IF bAutoStartPb AND ARbStnBasketAvailibilityRE[8].Q 	THEN ARbStnBasketInActivate[8] 	:= TRUE; ARsStnBasketInTime[8] := DSLocalSystemTimeML.sCurrentDateTime;
ARiStnBasketProductRecipeBuffer[8] 	:= DSStnBasketInfo[8].iProductRecipeNo; ARsStnBasketNoBuffer[8] 	:= DSStnBasketInfo[8].sReservedInt; 	END_IF

IF bAutoStartPb AND ARbStnBasketAvailibilityFE[8].Q 	THEN ARbStnBasketOutActivate[8] 	:= TRUE; ARsStnBasketOutTime[8] := DSLocalSystemTimeML.sCurrentDateTime; 	END_IF

IF bAutoStartPb AND ARbStnBasketAvailibilityRE[9].Q 	THEN ARbStnBasketInActivate[9] 	:= TRUE; ARsStnBasketInTime[9] := DSLocalSystemTimeML.sCurrentDateTime;
ARiStnBasketProductRecipeBuffer[9] 	:= DSStnBasketInfo[9].iProductRecipeNo; ARsStnBasketNoBuffer[9] 	:= DSStnBasketInfo[9].sReservedInt; 	END_IF

IF bAutoStartPb AND ARbStnBasketAvailibilityFE[9].Q 	THEN ARbStnBasketOutActivate[9] 	:= TRUE; ARsStnBasketOutTime[9] := DSLocalSystemTimeML.sCurrentDateTime; 	END_IF

IF bAutoStartPb AND ARbStnBasketAvailibilityRE[10].Q 	THEN ARbStnBasketInActivate[10] 	:= TRUE; ARsStnBasketInTime[10] := DSLocalSystemTimeML.sCurrentDateTime;
ARiStnBasketProductRecipeBuffer[10] 	:= DSStnBasketInfo[10].iProductRecipeNo; ARsStnBasketNoBuffer[10] 	:= DSStnBasketInfo[10].sReservedInt; 	END_IF

IF bAutoStartPb AND ARbStnBasketAvailibilityFE[10].Q 	THEN ARbStnBasketOutActivate[10] 	:= TRUE; ARsStnBasketOutTime[10] := DSLocalSystemTimeML.sCurrentDateTime; 	END_IF

//IF bAutoStartPb AND ARbStnBasketAvailibilityRE[11].Q 	THEN ARbStnBasketInActivate[11] 	:= TRUE; ARsStnBasketInTime[11] := DSLocalSystemTimeML.sCurrentDateTime;
//ARiStnBasketProductRecipeBuffer[11] 	:= DSStnBasketInfo[11].iProductRecipeNo; ARsStnBasketNoBuffer[11] 	:= DSStnBasketInfo[11].sReservedInt; 	END_IF

//IF bAutoStartPb AND ARbStnBasketAvailibilityFE[11].Q 	THEN ARbStnBasketOutActivate[11] 	:= TRUE; ARsStnBasketOutTime[11] := DSLocalSystemTimeML.sCurrentDateTime; 	END_IF

//IF bAutoStartPb AND ARbStnBasketAvailibilityRE[12].Q 	THEN ARbStnBasketInActivate[12] 	:= TRUE; ARsStnBasketInTime[12] := DSLocalSystemTimeML.sCurrentDateTime;
//ARiStnBasketProductRecipeBuffer[12] 	:= DSStnBasketInfo[12].iProductRecipeNo; ARsStnBasketNoBuffer[12] 	:= DSStnBasketInfo[12].sReservedInt; 	END_IF

//IF bAutoStartPb AND ARbStnBasketAvailibilityFE[12].Q 	THEN ARbStnBasketOutActivate[12] 	:= TRUE; ARsStnBasketOutTime[12] := DSLocalSystemTimeML.sCurrentDateTime; 	END_IF



IF bAutoStartPb AND ARtLdNotBasketAvailibility[1].Q 	THEN ARbLdBasketInActivate[1] 	:= FALSE;  	END_IF

IF bAutoStartPb AND ARtUldNotBasketAvailibility[1].Q 	THEN ARbUldBasketInActivate[1] 	:= FALSE; 	END_IF
//IF bAutoStartPb AND ARtUldNotBasketAvailibility[2].Q 	THEN ARbUldBasketInActivate[2] 	:= FALSE; 	END_IF

IF bAutoStartPb AND ARtStnNotBasketAvailibility[1].Q 	THEN ARbStnBasketInActivate[1] 	:= FALSE; 	ARbStnBasketOutActivate[1] 	:= FALSE; 	END_IF
IF bAutoStartPb AND ARtStnNotBasketAvailibility[2].Q 	THEN ARbStnBasketInActivate[2] 	:= FALSE; 	ARbStnBasketOutActivate[2] 	:= FALSE; 	END_IF
IF bAutoStartPb AND ARtStnNotBasketAvailibility[3].Q 	THEN ARbStnBasketInActivate[3] 	:= FALSE; 	ARbStnBasketOutActivate[3] 	:= FALSE; 	END_IF
IF bAutoStartPb AND ARtStnNotBasketAvailibility[4].Q 	THEN ARbStnBasketInActivate[4] 	:= FALSE; 	ARbStnBasketOutActivate[4] 	:= FALSE; 	END_IF
IF bAutoStartPb AND ARtStnNotBasketAvailibility[5].Q 	THEN ARbStnBasketInActivate[5] 	:= FALSE; 	ARbStnBasketOutActivate[5] 	:= FALSE; 	END_IF
IF bAutoStartPb AND ARtStnNotBasketAvailibility[6].Q 	THEN ARbStnBasketInActivate[6] 	:= FALSE; 	ARbStnBasketOutActivate[6] 	:= FALSE; 	END_IF
IF bAutoStartPb AND ARtStnNotBasketAvailibility[7].Q 	THEN ARbStnBasketInActivate[7] 	:= FALSE; 	ARbStnBasketOutActivate[7] 	:= FALSE; 	END_IF
IF bAutoStartPb AND ARtStnNotBasketAvailibility[8].Q 	THEN ARbStnBasketInActivate[8] 	:= FALSE; 	ARbStnBasketOutActivate[8] 	:= FALSE; 	END_IF
IF bAutoStartPb AND ARtStnNotBasketAvailibility[9].Q 	THEN ARbStnBasketInActivate[9] 	:= FALSE; 	ARbStnBasketOutActivate[9] 	:= FALSE; 	END_IF
IF bAutoStartPb AND ARtStnNotBasketAvailibility[10].Q 	THEN ARbStnBasketInActivate[10] 	:= FALSE; 	ARbStnBasketOutActivate[10] 	:= FALSE; 	END_IF
//IF bAutoStartPb AND ARtStnNotBasketAvailibility[11].Q 	THEN ARbStnBasketInActivate[11] 	:= FALSE; 	ARbStnBasketOutActivate[11] 	:= FALSE; 	END_IF
//IF bAutoStartPb AND ARtStnNotBasketAvailibility[12].Q 	THEN ARbStnBasketInActivate[12] 	:= FALSE; 	ARbStnBasketOutActivate[12] 	:= FALSE; 	END_IF

END_PROGRAM

// ---- POUs/MainProgram/DataManagement_Barcode/Log_Configuration.TcPOU
PROGRAM Log_Configuration
VAR
	fb1_dataLog: FB_jx_DataLog;
	fb2_dataLog: FB_jx_DataLog;
	fb3_dataLog: FB_jx_DataLog;
	fb4_dataLog: FB_jx_DataLog;
	fb5_dataLog: FB_jx_DataLog;
	fb6_dataLog: FB_jx_DataLog;
	fb7_dataLog: FB_jx_DataLog;
	fb8_dataLog: FB_jx_DataLog;
	fb9_dataLog: FB_jx_DataLog;
	fb10_dataLog: FB_jx_DataLog;
	(*fb11_dataLog: FB_jx_DataLog;
	fb12_dataLog: FB_jx_DataLog;*)
	fb13_dataLog: FB_jx_DataLog;

	tStn1		: TON;
	tStn2		: TON;
	tStn3		: TON;
	tStn4		: TON;
	tStn5		: TON;
	tStn6		: TON;
	tStn7		: TON;
	tStn8		: TON;
	tStn9		: TON;
	tStn10		: TON;
	tStn11		: TON;
	tStn12		: TON;
	tStn13		: TON;
	uldONtrig	:TON;

	test1		:BOOL;
	test2		:BOOL;
	test3		:BOOL;
	test4		:BOOL;
	test5		:BOOL;
	test6		:BOOL;
	test7		:BOOL;
	test8		:BOOL;
	test9		:BOOL;
	test10		:BOOL;
	test11		:BOOL;
	test12		:BOOL;
	test13		:BOOL;
	test14		:BOOL;
	R_TRIG1	:R_TRIG;
	R_TRIG2	:R_TRIG;
	R_TRIG3	:R_TRIG;

	reset		: BOOL;
	start			: BOOL;
	busy		: BOOL;
	Done		: BOOL;
	write			:BOOL;
	write_done	:BOOL;
	ErrMsg		: STRING;

	tsTimeNow: TIMESTRUCT;


	fbFileRename    : FB_FileRename;
	sNetId          : T_AmsNetId;
        sOldName                : T_MaxString;
        sNewName                : T_MaxString;
        ePath           : E_OpenPath := PATH_GENERIC;          (* Default: generic file path*)
        bExecute                : BOOL;
        tTimeout                : TIME;

	start1: BOOL;
	sPath: STRING;
	sPath1: STRING;
	sNameFile: STRING(255);
	sNameFile1: STRING(255);
	sNameFile2: STRING(255);
	sNameFile3: STRING(255);
	sNameFile4: STRING(255);
	sNameFile5: STRING(255);	(*  *)
	sNameFile6: STRING(255);	(*  *)
	sNameFile7: STRING(255);	(*  *)
	sNameFile8: STRING(255);	(*  *)
	sNameFile9: STRING(255);	(*  *)
	sNameFile10: STRING(255);	(*  *)
	sNameFile11: STRING(255);	(*  *)

	sTimeNow	:STRING;
	RE_BasketCount :R_TRIG;
	iBasketCount:INT;

	bRename: BOOL;
END_VAR

(*
(*All station, only after Remaining timer less than 10 sec, trigger Write CSV*)

tStn1(IN:=ARDsStnSeqProcessCtrl[1].Out_iTotalProcessTimeEV >0 AND ARDsStnSeqProcessCtrl[1].Out_iTotalProcessTimeEV <10 , PT:=T#1s , Q=> , ET=> );
tStn2(IN:=ARDsStnSeqProcessCtrl[2].Out_iTotalProcessTimeEV >0 AND ARDsStnSeqProcessCtrl[2].Out_iTotalProcessTimeEV <10 , PT:=T#1s , Q=> , ET=> );
tStn3(IN:=ARDsStnSeqProcessCtrl[3].Out_iTotalProcessTimeEV >0 AND ARDsStnSeqProcessCtrl[3].Out_iTotalProcessTimeEV <10 , PT:=T#1s , Q=> , ET=> );
tStn4(IN:=ARDsStnSeqProcessCtrl[4].Out_iTotalProcessTimeEV >0 AND ARDsStnSeqProcessCtrl[4].Out_iTotalProcessTimeEV <10  , PT:=T#1s , Q=> , ET=> );
tStn5(IN:=ARDsStnSeqProcessCtrl[5].Out_iTotalProcessTimeEV >0 AND ARDsStnSeqProcessCtrl[5].Out_iTotalProcessTimeEV <10 , PT:=T#1s , Q=> , ET=> );
tStn6(IN:=ARDsStnSeqProcessCtrl[6].Out_iTotalProcessTimeEV >0 AND ARDsStnSeqProcessCtrl[6].Out_iTotalProcessTimeEV <10 , PT:=T#1s , Q=> , ET=> );
tStn7(IN:=ARDsStnSeqProcessCtrl[7].Out_iTotalProcessTimeEV >0 AND ARDsStnSeqProcessCtrl[7].Out_iTotalProcessTimeEV <10 , PT:=T#1s , Q=> , ET=> );
tStn8(IN:=ARDsStnSeqProcessCtrl[8].Out_iTotalProcessTimeEV >0 AND ARDsStnSeqProcessCtrl[8].Out_iTotalProcessTimeEV <10 , PT:=T#1s , Q=> , ET=> );
tStn9(IN:=ARDsStnSeqProcessCtrl[9].Out_iTotalProcessTimeEV >0 AND ARDsStnSeqProcessCtrl[9].Out_iTotalProcessTimeEV <10 , PT:=T#1s, Q=> , ET=> );
tStn10(IN:=ARDsStnSeqProcessCtrl[10].Out_iTotalProcessTimeEV >0 AND ARDsStnSeqProcessCtrl[10].Out_iTotalProcessTimeEV <10 , PT:=T#1s , Q=> , ET=> );
tStn11(IN:=ARDsStnSeqProcessCtrl[11].Out_iTotalProcessTimeEV >0 AND ARDsStnSeqProcessCtrl[11].Out_iTotalProcessTimeEV <10 , PT:=T#1s , Q=> , ET=> );
tStn12(IN:=ARDsStnSeqProcessCtrl[12].Out_iTotalProcessTimeEV >0 AND ARDsStnSeqProcessCtrl[12].Out_iTotalProcessTimeEV <10 , PT:=T#1s , Q=> , ET=> );



(*Create a counter to give a number basket count at the File Name*)

sStn1tittle := CONCAT('-',DSStnBasketInfo[1].ARsBarcodeData[1]);
sStn1tittle := CONCAT(DSStnBasketInfo[1].ARsBarcodeData[2],sStn1tittle);
sStn1tittle := CONCAT('-',sStn1tittle);
sStn1tittle := CONCAT(DSStnBasketInfo[1].ARsBarcodeData[3],sStn1tittle);
sStn1tittle := CONCAT('-',sStn1tittle);
sStn1tittle := CONCAT(DSStnBasketInfo[1].sReservedInt,sStn1tittle);



fb1_dataLog(
	bActivate:= DSStnBasketInfo[1].bAvailibility AND  (tStn1.Q OR GeneratorComparison.ARUpdate_bIntAddress[1]) ,
	FolderDirectory:= 'C:\JKS\report_csv',
	sFileName:= sStn1tittle,
	Tittle := sStn1tittle,
	nNumberOfData:= 50,		(*Max 1000*)
	a_sDataLog_In:= a1_dataLink,
	TimeInterval:= Interval_5s,
	sCsvSeperator:= ',',
	tsTimeNow:=CurrentTime,
	enFIleType:= TXT, 			(*or	 enFIleType:= TXT, 		two option*)
	sMsg=> );


sStn2tittle := CONCAT('-',DSStnBasketInfo[2].ARsBarcodeData[1]);
sStn2tittle := CONCAT(DSStnBasketInfo[2].ARsBarcodeData[2],sStn2tittle);
sStn2tittle := CONCAT('-',sStn2tittle);
sStn2tittle := CONCAT(DSStnBasketInfo[2].ARsBarcodeData[3],sStn2tittle);
sStn2tittle := CONCAT('-',sStn2tittle);
sStn2tittle := CONCAT(DSStnBasketInfo[2].sReservedInt,sStn2tittle);

fb2_dataLog(
	bActivate:= DSStnBasketInfo[2].bAvailibility AND  (tStn2.Q OR GeneratorComparison.ARUpdate_bIntAddress[2]) ,
	FolderDirectory:= 'C:\JKS\report_csv',
	sFileName:= sStn2tittle,
	Tittle := sStn2tittle,
	nNumberOfData:= 50,		(*Max 1000*)
	a_sDataLog_In:= a2_dataLink,
	TimeInterval:= Interval_5s,
	sCsvSeperator:= ',',
	tsTimeNow:=CurrentTime,
	enFIleType:= TXT, 			(*or	 enFIleType:= TXT, 		two option*)
	sMsg=> );


sStn3tittle := CONCAT('-',DSStnBasketInfo[3].ARsBarcodeData[1]);
sStn3tittle := CONCAT(DSStnBasketInfo[3].ARsBarcodeData[2],sStn3tittle);
sStn3tittle := CONCAT('-',sStn3tittle);
sStn3tittle := CONCAT(DSStnBasketInfo[3].ARsBarcodeData[3],sStn3tittle);
sStn3tittle := CONCAT('-',sStn3tittle);
sStn3tittle := CONCAT(DSStnBasketInfo[3].sReservedInt,sStn3tittle);


fb3_dataLog(
	bActivate:= DSStnBasketInfo[3].bAvailibility AND  (tStn3.Q OR GeneratorComparison.ARUpdate_bIntAddress[3]) ,
	FolderDirectory:= 'C:\JKS\report_csv',
	sFileName:= sStn3tittle,
	Tittle := sStn3tittle,
	nNumberOfData:= 50,		(*Max 1000*)
	a_sDataLog_In:= a3_dataLink,
	TimeInterval:= Interval_5s,
	sCsvSeperator:= ',',
	tsTimeNow:=CurrentTime,
	enFIleType:= TXT, 			(*or	 enFIleType:= TXT, 		two option*)
	sMsg=> );


sStn4tittle := CONCAT('-',DSStnBasketInfo[4].ARsBarcodeData[1]);
sStn4tittle := CONCAT(DSStnBasketInfo[4].ARsBarcodeData[2],sStn4tittle);
sStn4tittle := CONCAT('-',sStn4tittle);
sStn4tittle := CONCAT(DSStnBasketInfo[4].ARsBarcodeData[3],sStn4tittle);
sStn4tittle := CONCAT('-',sStn4tittle);
sStn4tittle := CONCAT(DSStnBasketInfo[4].sReservedInt,sStn4tittle);


fb4_dataLog(
	bActivate:= DSStnBasketInfo[4].bAvailibility AND  tStn4.Q ,
	FolderDirectory:= 'C:\JKS\report_csv',
	sFileName:= sStn4tittle,
	Tittle := sStn4tittle,
	nNumberOfData:= 50,		(*Max 1000*)
	a_sDataLog_In:= a4_dataLink,
	TimeInterval:= Interval_5s,
	sCsvSeperator:= ',',
	tsTimeNow:=CurrentTime,
	enFIleType:= TXT, 			(*or	 enFIleType:= TXT, 		two option*)
	sMsg=> );


sStn5tittle := CONCAT('-',DSStnBasketInfo[5].ARsBarcodeData[1]);
sStn5tittle := CONCAT(DSStnBasketInfo[5].ARsBarcodeData[2],sStn5tittle);
sStn5tittle := CONCAT('-',sStn5tittle);
sStn5tittle := CONCAT(DSStnBasketInfo[5].ARsBarcodeData[3],sStn5tittle);
sStn5tittle := CONCAT('-',sStn5tittle);
sStn5tittle := CONCAT(DSStnBasketInfo[5].sReservedInt,sStn5tittle);


fb5_dataLog(
	bActivate:= DSStnBasketInfo[5].bAvailibility AND  (tStn5.Q OR GeneratorComparison.ARUpdate_bIntAddress[5]) ,
	FolderDirectory:= 'C:\JKS\report_csv',
	sFileName:= sStn5tittle,
	Tittle := sStn5tittle,
	nNumberOfData:= 50,		(*Max 1000*)
	a_sDataLog_In:= a5_dataLink,
	TimeInterval:= Interval_5s,
	sCsvSeperator:= ',',
	tsTimeNow:=CurrentTime,
	enFIleType:= TXT, 			(*or	 enFIleType:= TXT, 		two option*)
	sMsg=> );


sStn6tittle := CONCAT('-',DSStnBasketInfo[6].ARsBarcodeData[1]);
sStn6tittle := CONCAT(DSStnBasketInfo[6].ARsBarcodeData[2],sStn6tittle);
sStn6tittle := CONCAT('-',sStn6tittle);
sStn6tittle := CONCAT(DSStnBasketInfo[6].ARsBarcodeData[3],sStn6tittle);
sStn6tittle := CONCAT('-',sStn6tittle);
sStn6tittle := CONCAT(DSStnBasketInfo[6].sReservedInt,sStn6tittle);


fb6_dataLog(
	bActivate:= DSStnBasketInfo[6].bAvailibility AND  tStn6.Q ,
	FolderDirectory:= 'C:\JKS\report_csv',
	sFileName:= sStn6tittle,
	Tittle := sStn6tittle,
	nNumberOfData:= 50,		(*Max 1000*)
	a_sDataLog_In:= a6_dataLink,
	TimeInterval:= Interval_5s,
	sCsvSeperator:= ',',
	tsTimeNow:=CurrentTime,
	enFIleType:= TXT, 			(*or	 enFIleType:= TXT, 		two option*)
	sMsg=> );


sStn7tittle := CONCAT('-',DSStnBasketInfo[7].ARsBarcodeData[1]);
sStn7tittle := CONCAT(DSStnBasketInfo[7].ARsBarcodeData[2],sStn7tittle);
sStn7tittle := CONCAT('-',sStn7tittle);
sStn7tittle := CONCAT(DSStnBasketInfo[7].ARsBarcodeData[3],sStn7tittle);
sStn7tittle := CONCAT('-',sStn7tittle);
sStn7tittle := CONCAT(DSStnBasketInfo[7].sReservedInt,sStn7tittle);

fb7_dataLog(
	bActivate:= DSStnBasketInfo[7].bAvailibility AND  (tStn7.Q OR GeneratorComparison.ARUpdate_bIntAddress[7]) ,
	FolderDirectory:= 'C:\JKS\report_csv',
	sFileName:= sStn7tittle,
	Tittle := sStn7tittle,
	nNumberOfData:= 50,		(*Max 1000*)
	a_sDataLog_In:= a7_dataLink,
	TimeInterval:= Interval_5s,
	sCsvSeperator:= ',',
	tsTimeNow:=CurrentTime,
	enFIleType:= TXT, 			(*or	 enFIleType:= TXT, 		two option*)
	sMsg=> );


sStn8tittle := CONCAT('-',DSStnBasketInfo[8].ARsBarcodeData[1]);
sStn8tittle := CONCAT(DSStnBasketInfo[8].ARsBarcodeData[2],sStn8tittle);
sStn8tittle := CONCAT('-',sStn8tittle);
sStn8tittle := CONCAT(DSStnBasketInfo[8].ARsBarcodeData[3],sStn8tittle);
sStn8tittle := CONCAT('-',sStn8tittle);
sStn8tittle := CONCAT(DSStnBasketInfo[8].sReservedInt,sStn8tittle);

fb8_dataLog(
	bActivate:= DSStnBasketInfo[8].bAvailibility AND  tStn8.Q,
	FolderDirectory:= 'C:\JKS\report_csv',
	sFileName:= sStn8tittle,
	Tittle := sStn8tittle,
	nNumberOfData:= 50,		(*Max 1000*)
	a_sDataLog_In:= a8_dataLink,
	TimeInterval:= Interval_5s,
	sCsvSeperator:= ',',
	tsTimeNow:=CurrentTime,
	enFIleType:= TXT, 			(*or	 enFIleType:= TXT, 		two option*)
	sMsg=> );


sStn9tittle := CONCAT('-',DSStnBasketInfo[9].ARsBarcodeData[1]);
sStn9tittle := CONCAT(DSStnBasketInfo[9].ARsBarcodeData[2],sStn9tittle);
sStn9tittle := CONCAT('-',sStn9tittle);
sStn9tittle := CONCAT(DSStnBasketInfo[9].ARsBarcodeData[3],sStn9tittle);
sStn9tittle := CONCAT('-',sStn9tittle);
sStn9tittle := CONCAT(DSStnBasketInfo[9].sReservedInt,sStn9tittle);

fb9_dataLog(
	bActivate:= DSStnBasketInfo[9].bAvailibility AND  tStn9.Q ,
	FolderDirectory:= 'C:\JKS\report_csv',
	sFileName:= sStn9tittle,
	Tittle := sStn9tittle,
	nNumberOfData:= 50,		(*Max 1000*)
	a_sDataLog_In:= a9_dataLink,
	TimeInterval:= Interval_5s,
	sCsvSeperator:= ',',
	tsTimeNow:=CurrentTime,
	enFIleType:= TXT, 			(*or	 enFIleType:= TXT, 		two option*)
	sMsg=> );


sStn10tittle := CONCAT('-',DSStnBasketInfo[10].ARsBarcodeData[1]);
sStn10tittle := CONCAT(DSStnBasketInfo[10].ARsBarcodeData[2],sStn10tittle);
sStn10tittle := CONCAT('-',sStn10tittle);
sStn10tittle := CONCAT(DSStnBasketInfo[10].ARsBarcodeData[3],sStn10tittle);
sStn10tittle := CONCAT('-',sStn10tittle);
sStn10tittle := CONCAT(DSStnBasketInfo[10].sReservedInt,sStn10tittle);

fb10_dataLog(
	bActivate:=DSStnBasketInfo[10].bAvailibility AND  tStn10.Q,
	FolderDirectory:= 'C:\JKS\report_csv',
	sFileName:= sStn10tittle,
	Tittle := sStn10tittle,
	nNumberOfData:= 50,		(*Max 1000*)
	a_sDataLog_In:= a10_dataLink,
	TimeInterval:= Interval_5s,
	sCsvSeperator:= ',',
	tsTimeNow:=CurrentTime,
	enFIleType:= TXT, 			(*or	 enFIleType:= TXT, 		two option*)
	sMsg=> );

(*
sStn11tittle := CONCAT('-',DSStnBasketInfo[11].ARsBarcodeData[1]);
sStn11tittle := CONCAT(DSStnBasketInfo[11].ARsBarcodeData[2],sStn11tittle);
sStn11tittle := CONCAT('-',sStn11tittle);
sStn11tittle := CONCAT(DSStnBasketInfo[11].ARsBarcodeData[3],sStn11tittle);
sStn11tittle := CONCAT('-',sStn11tittle);
sStn11tittle := CONCAT(DSStnBasketInfo[11].sReservedInt,sStn11tittle);

fb11_dataLog(
	bActivate:=DSStnBasketInfo[11].bAvailibility AND  tStn11.Q ,
	FolderDirectory:= 'C:\JKS\report_csv',
	sFileName:= sStn11tittle,
	Tittle := sStn11tittle,
	nNumberOfData:= 50,		(*Max 1000*)
	a_sDataLog_In:= a11_dataLink,
	TimeInterval:= Interval_5s,
	sCsvSeperator:= ',',
	tsTimeNow:=CurrentTime,
	enFIleType:= TXT, 			(*or	 enFIleType:= TXT, 		two option*)
	sMsg=> );

sStn12tittle := CONCAT('-',DSStnBasketInfo[12].ARsBarcodeData[1]);
sStn12tittle := CONCAT(DSStnBasketInfo[12].ARsBarcodeData[2],sStn12tittle);
sStn12tittle := CONCAT('-',sStn12tittle);
sStn12tittle := CONCAT(DSStnBasketInfo[12].ARsBarcodeData[3],sStn12tittle);
sStn12tittle := CONCAT('-',sStn12tittle);
sStn12tittle := CONCAT(DSStnBasketInfo[12].sReservedInt,sStn12tittle);

fb12_dataLog(
	bActivate:=DSStnBasketInfo[12].bAvailibility AND  tStn12.Q ,
	FolderDirectory:= 'C:\JKS\report_csv',
	sFileName:= sStn12tittle,
	Tittle := sStn12tittle,
	nNumberOfData:= 50,		(*Max 1000*)
	a_sDataLog_In:= a12_dataLink,
	TimeInterval:= Interval_5s,
	sCsvSeperator:= ',',
	tsTimeNow:=CurrentTime,
	enFIleType:= TXT, 			(*or	 enFIleType:= TXT, 		two option*)
	sMsg=> );
*)

(*
sStn13tittle := CONCAT('-',AR2sDSCv_UldConfirmBasketInfo[1,1].ARsBarcodeData[1]);
sStn13tittle := CONCAT(AR2sDSCv_UldConfirmBasketInfo[1,1].ARsBarcodeData[2],sStn13tittle);
sStn13tittle := CONCAT('-',sStn13tittle);
sStn13tittle := CONCAT(AR2sDSCv_UldConfirmBasketInfo[1,1].ARsBarcodeData[3],sStn13tittle);


fb13_dataLog(
	bActivate:= AR2sDSCv_UldConfirmBasketInfo[1,1].bAvailibility (*AND tStn12.Q*) OR test12 (*Trigger Bit when Arm in Down unhook pos*) ,
	FolderDirectory:= 'C:\JKS\report_csv',
	sFileName:= sStn13tittle,
	Tittle := sStn13tittle,
	nNumberOfData:= 50,		(*Max 1000*)
	a_sDataLog_In:= a12_dataLink,
	TimeInterval:= Interval_5s,
	sCsvSeperator:= ',',
	tsTimeNow:=CurrentTime,
	enFIleType:= TXT, 			(*or	 enFIleType:= TXT, 		two option*)
	sMsg=> );
*)

(*To complete the CSV file write at Unloading area*)
IF ARDSArmCtrl[2].AR3sbPositionCfm[3,1,8] OR test14 THEN

	sStn13tittle := CONCAT('-',DSArmBasketInfo[2].ARsBarcodeData[1]);
	sStn13tittle := CONCAT(DSArmBasketInfo[2].ARsBarcodeData[2],sStn13tittle);
	sStn13tittle := CONCAT('-',sStn13tittle);
	sStn13tittle := CONCAT(DSArmBasketInfo[2].ARsBarcodeData[3],sStn13tittle);
	sStn13tittle := CONCAT('-',sStn13tittle);
	sStn13tittle := CONCAT(DSArmBasketInfo[2].sReservedInt,sStn13tittle);

END_IF



(* Trigger bit when Unloading*)
tStn13(IN:=AR2sDSCv_UldConfirmBasketInfo[1,1].bAvailibility , PT:=T#1s , Q=> , ET=> );
R_TRIG1(CLK:=tStn13.Q  OR test13  , Q=> );

	IF R_TRIG1.Q  THEN
		start:=TRUE;
		ELSE
		start:=FALSE;
	END_IF


CurrentTime:=stGetCurrentTime.SysTime;

(*NOTE:-

1-sPath and sPath MUST SAME NAME, otherwise file will not overwrite*)

sPath:=CONCAT('C:\JKS\report_csv','\');
sPath:=CONCAT(sPath,sStn13tittle);
sPath:=CONCAT(sPath,'_');
sPath:=CONCAT(sPath,F_jx_TS_TO_DATE_STRING_1(CurrentTime, '_'));
sPath:=CONCAT(sPath,'.cs_');


sPath1:=CONCAT('C:\JKS\report_csv','\');
sPath1:=CONCAT(sPath1,sStn13tittle);
sPath1:=CONCAT(sPath1,'_');
sPath1:=CONCAT(sPath1,F_jx_TS_TO_DATE_STRING_1(CurrentTime, '_'));
sPath1:=CONCAT(sPath1,'.csv');

fbFileRename(
	sOldName:=sPath ,
	sNewName:=sPath1 ,
	ePath:= PATH_GENERIC,
	bExecute:=bRename OR start);
*)

END_PROGRAM

// ---- FBs/B_JKS_CustomFB/fbDataLogCtrl/FB_jx_DataLog.TcPOU
FUNCTION_BLOCK FB_jx_DataLog
VAR_INPUT
	bActivate:BOOL;		(*Activate data logging*)
	FolderDirectory: T_MaxString;		(*Folder to save log file*)
	Tittle	: T_MaxString;
	sFileName: STRING:='DataLog';
	nNumberOfData:INT:=100;		(*number of data going to log*)
	a_sDataLog_In: ARRAY [1..100] OF ST_DataLog;		(*Log Data name and Value, in string form*)
	TimeInterval: En_TimeInterval:=Interval_1min;		(*Time interval for data logging *)
	sCsvSeperator:STRING:=',';		(*Seperator for Csv file*)
	tsTimeNow: TIMESTRUCT;		(*Time now*)
	enFIleType: En_LogFileType:=CSV;		(*2 Option: CSV ,  TXT*)
	bDirectWrite			: BOOL;
END_VAR
VAR_OUTPUT
	sMsg:STRING;
END_VAR
VAR
	nWriteLogState: INT;
	bTrigWri: BOOL;
	R_TRIG_Wri: R_TRIG;
	a_sDataLog: ARRAY [1..100] OF ST_DataLog;		(*Log Data name and Value, in string form*)
	tsTimeMoment: TIMESTRUCT;
	fbTimeTriggering: FB_TimeTriggering;
	fbWriteLog:FB_WriteLog;
END_VAR

(*
Create by: Jun Xian
Date: 28 May 2014
Modify: 21 Sep 2015

Purpose: 
1. Log data Into Csv file


Feature:
1. Selectable csv seperator.
2. Everyday using a new log file.
3. Selectable data log time interval.
4. Currently number of data support up to 1000 data. 
5. Log File can select save as .CSV or .TXT.

Limitation:
1. If data name > 50, maybe will cause some word missing.
*)
(*
IF bActivate  THEN
fbTimeTriggering(en_interval:= TimeInterval, tsTimeNow:= tsTimeNow, bTrigWriLog=> );
*)
IF bActivate  THEN
bTrigWri := TRUE;
ELSE
bTrigWri := FALSE;
END_IF

R_TRIG_Wri(CLK:= bTrigWri , Q=> );
IF R_TRIG_Wri.Q THEN		(*record the value at that moment*)
a_sDataLog:=a_sDataLog_In;
tsTimeMoment:=tsTimeNow;
END_IF

fbWriteLog(
	sFolderDirectory:= FolderDirectory,
	sTittle := Tittle,
	aDataLog:= a_sDataLog,
	sSeperator:= sCsvSeperator,
	tsTimeMoment:= tsTimeMoment,
	tsTimeNow:= tsTimeNow,
	bStartWri:= R_TRIG_Wri.Q,
	nNumOfData:= nNumberOfData,
	enFileType:= enFIleType,
	sFileName:= sFileName,
	sErrMsg=> sMsg);

END_FUNCTION_BLOCK

// ---- FBs/B_JKS_CustomFB/fbDataLogCtrl/FB_TimeTriggering.TcPOU
FUNCTION_BLOCK FB_TimeTriggering
VAR_INPUT
	en_interval: En_TimeInterval;
	tsTimeNow: TIMESTRUCT;
END_VAR
VAR_OUTPUT
	bTrigWriLog: BOOL;
END_VAR
VAR
	bTest: BOOL;
	wSecPrev: WORD;
END_VAR

IF tsTimeNow.wYear <> 1970 AND tsTimeNow.wYear <> 0 THEN

CASE en_interval OF

Interval_1s:
	IF (tsTimeNow.wSecond <> wSecPrev) THEN
		wSecPrev:=tsTimeNow.wSecond;
		bTrigWriLog:=TRUE;
	ELSE
		bTrigWriLog:=FALSE;
	END_IF

Interval_5s:
	IF (tsTimeNow.wSecond MOD 5 = 0) THEN
		bTrigWriLog:=TRUE;
	ELSE
		bTrigWriLog:=FALSE;
	END_IF

Interval_10s:
	IF (tsTimeNow.wSecond MOD 10 = 0) THEN
		bTrigWriLog:=TRUE;
	ELSE
		bTrigWriLog:=FALSE;
	END_IF

Interval_20s:
	IF (tsTimeNow.wSecond MOD 20 = 0) THEN
	bTrigWriLog:=TRUE;
	ELSE
		bTrigWriLog:=FALSE;
	END_IF

Interval_30s:
	IF (tsTimeNow.wSecond MOD 30 = 0) THEN
	bTrigWriLog:=TRUE;
	ELSE
		bTrigWriLog:=FALSE;
	END_IF

Interval_1min:
	IF (tsTimeNow.wSecond = 0) THEN
	bTrigWriLog:=TRUE;
	ELSE
		bTrigWriLog:=FALSE;
	END_IF

Interval_2min:
	IF (tsTimeNow.wSecond = 0) AND (tsTimeNow.wMinute MOD 2 = 0)THEN
	bTrigWriLog:=TRUE;
	ELSE
		bTrigWriLog:=FALSE;
	END_IF

Interval_5min:
	IF (tsTimeNow.wSecond = 0) AND (tsTimeNow.wMinute MOD 5 = 0)THEN
	bTrigWriLog:=TRUE;
	ELSE
		bTrigWriLog:=FALSE;
	END_IF

Interval_10min:
	IF (tsTimeNow.wSecond = 0) AND (tsTimeNow.wMinute MOD 10 = 0)THEN
	bTrigWriLog:=TRUE;
	ELSE
		bTrigWriLog:=FALSE;
	END_IF

Interval_15min:
	IF (tsTimeNow.wSecond = 0) AND (tsTimeNow.wMinute MOD 15 = 0)THEN
	bTrigWriLog:=TRUE;
	ELSE
		bTrigWriLog:=FALSE;
	END_IF

Interval_20min:
	IF (tsTimeNow.wSecond = 0) AND (tsTimeNow.wMinute MOD 20 = 0)THEN
	bTrigWriLog:=TRUE;
	ELSE
		bTrigWriLog:=FALSE;
	END_IF

Interval_30min:
	IF (tsTimeNow.wSecond = 0) AND (tsTimeNow.wMinute MOD 30 = 0)THEN
	bTrigWriLog:=TRUE;
	ELSE
		bTrigWriLog:=FALSE;
	END_IF

Interval_1h:
	IF (tsTimeNow.wSecond = 0) AND (tsTimeNow.wMinute = 0)THEN
	bTrigWriLog:=TRUE;
	ELSE
		bTrigWriLog:=FALSE;
	END_IF

Interval_2h:
	IF (tsTimeNow.wSecond = 0) AND (tsTimeNow.wMinute = 0) AND (tsTimeNow.wHour MOD 2 = 0)THEN
	bTrigWriLog:=TRUE;
	ELSE
		bTrigWriLog:=FALSE;
	END_IF


END_CASE

END_IF

END_FUNCTION_BLOCK

// ---- FBs/B_JKS_CustomFB/fbDataLogCtrl/FB_WriteLog.TcPOU
FUNCTION_BLOCK FB_WriteLog
VAR_INPUT
	sFolderDirectory: T_MaxString;
	sTittle : T_MaxString;
	aDataLog: ARRAY [1..100] OF ST_DataLog;
	sSeperator: STRING;
	tsTimeMoment: TIMESTRUCT;
	tsTimeNow: TIMESTRUCT;
	bStartWri: BOOL;		(*Been triggered when want start to write log*)
	nNumOfData: INT;
	enFileType: En_LogFileType;
	sFileName: STRING;
	nCurrWrite3: INT;
END_VAR
VAR_OUTPUT
	sErrMsg: STRING;
END_VAR
VAR
	sPath: T_MaxString;
	FB_FileOpen_Log: FB_FileOpen;
	nWriState: INT;
	sHeadline: T_MaxString;
	sHeadline2: T_MaxString;
	i: INT;
	FB_FilePuts_Log: FB_FilePuts;
	sValueLine: T_MaxString;
	FB_FileSeek_Log: FB_FileSeek;
	FB_FileClose_Log: FB_FileClose;
	nCurrWrite: INT := 1;
	bHeadLineDone: BOOL;
	bHeadlineDT: BOOL;
	bHeadlineDT2: BOOL;
	bHeadlineDT3: BOOL;
	bHeadlineDT4: BOOL;
	bDataDT: BOOL;
	bDataDone: BOOL;
	nCurDataWri: INT;
	i_1: INT;
	i_2: INT;
	i_3: INT;
	nCurrWrite2: INT;
	i_4: INT;
	i_5: INT;
	nCurrWrite4: INT;
END_VAR

sPath:=CONCAT(sFolderDirectory,'\');
sPath:=CONCAT(sPath,sFileName);
sPath:=CONCAT(sPath,'_');
sPath:=CONCAT(sPath,F_jx_TS_TO_DATE_STRING_1(tsTimeNow, '_'));
IF enFileType = CSV THEN
	sPath:=CONCAT(sPath,'.csv');
ELSIF enFileType = TXT THEN
	sPath:=CONCAT(sPath,'.cs_');
END_IF

FB_FileOpen_Log(
	sNetId:= ,
	sPathName:= sPath,
	nMode:= ,
	ePath:= PATH_GENERIC,
	bExecute:= ,
	tTimeout:= ,
	bBusy=> ,
	bError=> ,
	nErrId=> ,
	hFile=> );

FB_FilePuts_Log(
	sNetId:= ,
	hFile:= ,
	sLine:= ,
	bExecute:= ,
	tTimeout:= ,
	bBusy=> ,
	bError=> ,
	nErrId=> );

FB_FileSeek_Log(
	sNetId:= ,
	hFile:= ,
	nSeekPos:= ,
	eOrigin:= ,
	bExecute:= ,
	tTimeout:= ,
	bBusy=> ,
	bError=> ,
	nErrId=> );

FB_FileClose_Log(
	sNetId:= ,
	hFile:= ,
	bExecute:= ,
	tTimeout:= ,
	bBusy=> ,
	bError=> ,
	nErrId=> );

Act_WriLogSEQ();

ACTION act_PreapreDataValue:
IF bDataDT THEN
	sValueLine:=F_jx_TS_TO_TIME_STRING(tsTimeMoment);
	sValueLine:=CONCAT(sValueLine,sSeperator);
	(*sValueLine:=CONCAT(sValueLine,F_jx_TS_TO_TIME_STRING(tsTimeMoment));
	sValueLine:=CONCAT(sValueLine,sSeperator);*)
	bDataDT:=FALSE;
	nCurDataWri:=1;

END_IF

FOR i_1:= nCurDataWri TO 1000 DO
	IF i_1 > nNumOfData THEN
		sValueLine:=CONCAT(sValueLine,'$N');
		bDataDone:=TRUE;
EXIT;
	END_IF

	IF ((LEN(sValueLine)+LEN(sSeperator)+LEN(aDataLog[i_1].sValue))<240) THEN		(*T_MaxString is 250, 10 as buffer. the T-MaxString not full yet*)
		sValueLine:=CONCAT(sValueLine,aDataLog[i_1].sValue);
		sValueLine:=CONCAT(sValueLine,sSeperator);
	ELSE		(*T_MaxString is full*)
		bDataDone:=FALSE;
		nCurDataWri:=i_1;
EXIT;	(*T_MaxString is full, write 1st to CSV 1st*)
	END_IF

	IF (i_1 = 1000) THEN	(*Wrtie headline complete*)
		sValueLine:=CONCAT(sValueLine,'$N');
		bDataDone:=TRUE;
EXIT;	(*Write complete*)
	END_IF
END_FOR
END_ACTION

ACTION act_PreparingHeadline:
IF bHeadlineDT THEN		(*new day, need to prepare headline, just come from state 22*)
	(*sHeadline:=sTittle;
	sHeadline:=CONCAT(sHeadline,'$N'); *)


		nCurrWrite4:=1;

		FOR i_5:= nCurrWrite4 TO 7 DO
			IF i_5 > nNumOfData THEN
				sHeadline:=CONCAT(sHeadline,'$N');
				bHeadlineDT:=FALSE;

			EXIT;	(*Write complete*)
			END_IF

			IF ((LEN(sHeadline) + LEN(sSeperator) + LEN(aDataLog[i_5].sName4)) < 240 ) THEN		(*T_MaxString is 250, 10 as buffer. the T-MaxString not full yet*)
				sHeadline:=CONCAT(sHeadline, aDataLog[i_5].sName4);
				sHeadline:=CONCAT(sHeadline,sSeperator);
			ELSE		(*T_MaxString is full*)
				bHeadLineDone:=FALSE;
				nCurrWrite4:=i_5;
			EXIT;	(*T_MaxString is full, write 1st to CSV 1st*)
			END_IF

			IF (i_5 = 7) THEN	(*Wrtie headline complete*)
				sHeadline:=CONCAT(sHeadline,'$N');
				bHeadlineDT:=FALSE;
				bHeadlineDT2:=TRUE;
				nCurrWrite3:=1;
			EXIT;	(*Write complete*)
			END_IF
		END_FOR
END_IF

IF bHeadlineDT2 THEN

		FOR i_4:= nCurrWrite3 TO 7 DO
			IF i_4 > nNumOfData THEN
				sHeadline:=CONCAT(sHeadline,'$N');
				bHeadlineDT2:=FALSE;

			EXIT;	(*Write complete*)
			END_IF

			IF ((LEN(sHeadline) + LEN(sSeperator) + LEN(aDataLog[i_4].sName3)) < 240 ) THEN		(*T_MaxString is 250, 10 as buffer. the T-MaxString not full yet*)
				sHeadline:=CONCAT(sHeadline, aDataLog[i_4].sName3);
				sHeadline:=CONCAT(sHeadline,sSeperator);
			ELSE		(*T_MaxString is full*)
				bHeadLineDone:=FALSE;
				nCurrWrite3:=i_4;
			EXIT;	(*T_MaxString is full, write 1st to CSV 1st*)
			END_IF

			IF (i_4 = 7) THEN	(*Wrtie headline complete*)
				sHeadline:=CONCAT(sHeadline,'$N');
				bHeadlineDT2:=FALSE;
				bHeadlineDT3:=TRUE;
				nCurrWrite2:=1;
			EXIT;	(*Write complete*)
			END_IF
		END_FOR
END_IF

(*sHeadline:=CONCAT(sHeadline,'$N');*)

IF bHeadlineDT3 THEN

		FOR i_3:= nCurrWrite2 TO 50 DO
			IF i_3 > nNumOfData THEN
				sHeadline:=CONCAT(sHeadline,'$N');
				bHeadlineDT3:=FALSE;

			EXIT;	(*Write complete*)
			END_IF

			IF ((LEN(sHeadline) + LEN(sSeperator) + LEN(aDataLog[i_3].sName2)) < 240 ) THEN		(*T_MaxString is 250, 10 as buffer. the T-MaxString not full yet*)
				sHeadline:=CONCAT(sHeadline, aDataLog[i_3].sName2);
				sHeadline:=CONCAT(sHeadline,sSeperator);
			ELSE		(*T_MaxString is full*)
				bHeadLineDone:=FALSE;
				nCurrWrite2:=i_3;
			EXIT;	(*T_MaxString is full, write 1st to CSV 1st*)
			END_IF

			IF (i_3 = 50) THEN	(*Wrtie headline complete*)
				sHeadline:=CONCAT(sHeadline,'$N');
				bHeadlineDT3:=FALSE;
				nCurrWrite:=1;
			EXIT;	(*Write complete*)
			END_IF
		END_FOR

(*sHeadline:=CONCAT(sHeadline,'$N');*)(*comment by syafiq 190418*)

IF NOT (nCurrWrite2=i_3) THEN
	sHeadline:=CONCAT(sHeadline,'Time ');
	sHeadline:=CONCAT(sHeadline,sSeperator);
	bHeadlineDT:=FALSE;
	nCurrWrite:=1;
END_IF

END_IF

FOR i_2:= nCurrWrite TO 1000 DO
	IF i_2 > nNumOfData THEN
		sHeadline:=CONCAT(sHeadline,'$N');
		bHeadLineDone:=TRUE;
EXIT;	(*Write complete*)
	END_IF

	IF ((LEN(sHeadline) + LEN(sSeperator) + LEN(aDataLog[i_2].sName)) < 240 ) THEN		(*T_MaxString is 250, 10 as buffer. the T-MaxString not full yet*)
		sHeadline:=CONCAT(sHeadline, aDataLog[i_2].sName);
		sHeadline:=CONCAT(sHeadline,sSeperator);
	ELSE		(*T_MaxString is full*)
		bHeadLineDone:=FALSE;
		nCurrWrite:=i_2;
EXIT;	(*T_MaxString is full, write 1st to CSV 1st*)
	END_IF

	IF (i_2 = 1000) THEN	(*Wrtie headline complete*)
		sHeadline:=CONCAT(sHeadline,'$N');
		bHeadLineDone:=TRUE;
EXIT;	(*Write complete*)
	END_IF
END_FOR
END_ACTION

ACTION Act_WriLogSEQ:
CASE nWriState OF
0:		(*Iinitial State*)
	FB_FileOpen_Log(bExecute:= FALSE);
	FB_FileSeek_Log(bExecute:= FALSE);
	FB_FilePuts_Log(bExecute:= FALSE);
	FB_FileClose_Log(bExecute:= FALSE);
	
	IF bStartWri THEN
		sErrMsg:='';		(*clear error message*)
(*		bStartWri:=FALSE;*)
		nWriState:=10;
	END_IF

10:		(*Try to write as normal, file already exists*)
	FB_FileOpen_Log(bExecute:= FALSE);
	FB_FileOpen_Log(
		nMode:= FOPEN_MODEREAD OR FOPEN_MODEPLUS OR FOPEN_MODETEXT,
		ePath:= PATH_GENERIC,
		bExecute:= TRUE);

	IF FB_FileOpen_Log.bBusy THEN
		nWriState:=12;
	END_IF

12:		(*Determine whether got error, if error 1804 mean file not exist, need to create a new file*)
	IF NOT FB_FileOpen_Log.bBusy THEN
		IF NOT FB_FileOpen_Log.bError THEN
			nWriState:=14;		(*proceed to write data value*)
		ELSE
			IF (FB_FileOpen_Log.nErrId = 16#70C) THEN		(*no file, need to create a new one*)
			nWriState:=20;
			ELSE
			sErrMsg:='File Open Error [12]';
			nWriState:=0;
			END_IF
		END_IF
	END_IF


14:		(*File Seek, point to the end of file*)
	FB_FileSeek_Log(bExecute:= FALSE);
	FB_FileSeek_Log(
		hFile:= FB_FileOpen_Log.hFile,
		eOrigin:= SEEK_END,
		bExecute:= TRUE);
	
	IF FB_FileSeek_Log.bBusy THEN	(*Seek Fb start to run*)
	nWriState:=16;
	END_IF

16:
	IF NOT FB_FileSeek_Log.bBusy THEN
		IF NOT FB_FileSeek_Log.bError THEN	(*no error*)
bDataDT:=TRUE;
			nWriState:=40;		(*proceed to write *)
		ELSE	(*error*)
			sErrMsg:='File Seek error [16]';
			nWriState:=0;
		END_IF
	END_IF


20:		(*Open a new file, going to write the headline*)
	FB_FileOpen_Log(bExecute:= FALSE);
	FB_FileOpen_Log(
		nMode:= FOPEN_MODEAPPEND OR FOPEN_MODETEXT,
		ePath:= PATH_GENERIC,
		bExecute:= TRUE);
	IF FB_FileOpen_Log.bBusy THEN
		nWriState:=22;
	END_IF

22:		(*check whether got error*)
	IF NOT FB_FileOpen_Log.bBusy  THEN
		IF FB_FileOpen_Log.bError THEN		(*Error*)
			sErrMsg:='File Open error [22]';
			nWriState:=0;
		ELSE		(*no error, go to state 30*)
			nWriState:=30;
bHeadlineDT:=TRUE;
		END_IF

	END_IF


30:		(*Write Headline to Csv	|| Preparing Headline*)
sHeadline:='';
	act_PreparingHeadline();
	FB_FilePuts_Log(bExecute:= FALSE);
	FB_FilePuts_Log(
		hFile:= FB_FileOpen_Log.hFile,
		sLine:= sHeadline,
		bExecute:= TRUE);
	IF FB_FilePuts_Log.bBusy THEN		(*FB start to work*)
		nWriState:=32;
	END_IF

32:
	IF NOT FB_FilePuts_Log.bBusy THEN	(*Fb Done*)
		IF NOT FB_FilePuts_Log.bError THEN	(*no error*)

IF bHeadLineDone THEN	(*Writing headline is complete, can go to write data state*)
nWriState:=40;		(*proceed to write value*)
bDataDT:=TRUE;
ELSE
nWriState:=30;		(*continue to write headline*)
END_IF

		ELSE		(*got error*)
		sErrMsg:='Write Headline Error[32]';
		nWriState:=0;
		END_IF
	END_IF

40:		(*Write data value into csv*)
sValueLine:='';
	act_PreapreDataValue();
	FB_FilePuts_Log(bExecute:= FALSE);
	FB_FilePuts_Log(
		hFile:= FB_FileOpen_Log.hFile,
		sLine:= sValueLine,
		bExecute:= TRUE);
	IF FB_FilePuts_Log.bBusy THEN		(*FB start to work*)
		nWriState:=42;
	END_IF

42:
	IF NOT FB_FilePuts_Log.bBusy THEN
		IF NOT FB_FilePuts_Log.bError THEN	(*no error*)

IF bDataDone THEN		(*write data complete, proceed to close state*)
nWriState:=50;		(*proceed to close file*)
ELSE		(*data not finish write*)
nWriState:=40;		(*continue write data*)
END_IF

		ELSE		(*error*)
			sErrMsg:='Write Value Error[42]';
			nWriState:=0;
		END_IF
	END_IF

50:		(*Close file state*)
	FB_FileClose_Log(bExecute:= FALSE);
	FB_FileClose_Log(
		hFile:= FB_FileOpen_Log.hFile,
		bExecute:= TRUE);
	IF FB_FileClose_Log.bBusy THEN
		nWriState:=52;
	END_IF

52:
	IF NOT FB_FileClose_Log.bBusy THEN
		IF FB_FileClose_Log.bError THEN	(*error*)
		sErrMsg:='File CloseError[52]';
		nWriState:=0;	(*no matter how will goes back to initial state*)
		ELSE	(*no error*)
		nWriState:=0;	(*no matter how will goes back to initial state*)
		END_IF
	END_IF

END_CASE
END_ACTION

END_FUNCTION_BLOCK

// ---- FBs/B_JKS_CustomFB/fbDataLogCtrl/F_jx_TS_TO_DATE_STRING_1.TcPOU
FUNCTION F_jx_TS_TO_DATE_STRING_1 : STRING
VAR_INPUT
	ts_TimeNow: TIMESTRUCT;
	sSeperator: STRING := '/';
END_VAR
VAR
	sDate: STRING;
END_VAR

sDate:='';
sDate:=CONCAT(sDate,WORD_TO_STRING(ts_TimeNow.wYear));
IF ts_TimeNow.wMonth < 10 THEN	(**)
	sDate:=CONCAT(sDate,'0');
	sDate:=CONCAT(sDate,WORD_TO_STRING(ts_TimeNow.wMonth));
ELSE
	sDate:=CONCAT(sDate,WORD_TO_STRING(ts_TimeNow.wMonth));
END_IF

IF ts_TimeNow.wDay < 10 THEN
	sDate:=CONCAT(sDate,'0');
	sDate:=CONCAT(sDate,WORD_TO_STRING(ts_TimeNow.wDay));
ELSE
	sDate:=CONCAT(sDate,WORD_TO_STRING(ts_TimeNow.wDay));
END_IF
F_jx_TS_TO_DATE_STRING_1:=sDate;

END_FUNCTION

// ---- FBs/B_JKS_CustomFB/fbDataLogCtrl/F_jx_TS_TO_TIME_STRING.TcPOU
FUNCTION F_jx_TS_TO_TIME_STRING : STRING
VAR_INPUT
	ts_TimeNow: TIMESTRUCT;
END_VAR
VAR
	sTime:STRING;
	sSeperator: STRING := ':';
END_VAR

sTime:='';
IF ts_TimeNow.wHour < 10 THEN	(*Hour*)
sTime:=CONCAT(sTime,'0');
sTime:=CONCAT(sTime,WORD_TO_STRING(ts_TimeNow.wHour));
ELSE
sTime:=CONCAT(sTime,WORD_TO_STRING(ts_TimeNow.wHour));
END_IF

sTime:=CONCAT(sTime,sSeperator);

IF ts_TimeNow.wMinute < 10 THEN	(*Minute*)
sTime:=CONCAT(sTime,'0');
sTime:=CONCAT(sTime,WORD_TO_STRING(ts_TimeNow.wMinute));
ELSE
sTime:=CONCAT(sTime,WORD_TO_STRING(ts_TimeNow.wMinute));
END_IF

sTime:=CONCAT(sTime,sSeperator);

IF ts_TimeNow.wSecond < 10 THEN	(*Minute*)
sTime:=CONCAT(sTime,'0');
sTime:=CONCAT(sTime,WORD_TO_STRING(ts_TimeNow.wSecond));
ELSE
sTime:=CONCAT(sTime,WORD_TO_STRING(ts_TimeNow.wSecond));
END_IF

F_jx_TS_TO_TIME_STRING:=sTime;

END_FUNCTION

// ---- POUs/MainProgram/DataManagement_Barcode/Log_Management.TcPOU
PROGRAM Log_Management
VAR

END_VAR

;
(*
(*

a2_dataLink[1].sName4:='';
a2_dataLink[2].sName4:='Operator';
a2_dataLink[3].sName4:='Loading ID';
a2_dataLink[4].sName4:='Unloading ID';
a2_dataLink[5].sName4:='Product Recipe Number';
a2_dataLink[6].sName4:='Product Recipe Description';
a2_dataLink[7].sName4:='Load Number';
*)

a1_dataLink[1].sName4:='';
a1_dataLink[2].sName4:='Operator';
a1_dataLink[3].sName4:='LD ID';
a1_dataLink[4].sName4:='ULD ID';
a1_dataLink[5].sName4:='Pro Recipe No';
a1_dataLink[6].sName4:='Pro Recipe Dscrp';
a1_dataLink[7].sName4:='LD No';


a1_dataLink[1].sName3:='';
a1_dataLink[2].sName3:=sUserName;
a1_dataLink[3].sName3:='1';
a1_dataLink[4].sName3:='1';
a1_dataLink[5].sName3:=INT_TO_STRING(DSStnBasketInfo[1].iProductRecipeNo);
a1_dataLink[6].sName3:=DSStnBasketInfo[1].sProgramDescription;
a1_dataLink[7].sName3:=INT_TO_STRING(iProgBatchTotal);


a1_dataLink[1].sName2:='';
a1_dataLink[2].sName2:='N/A';
a1_dataLink[3].sName2:='N/A';
a1_dataLink[4].sName2:='N/A';
a1_dataLink[5].sName2:='N/A';
a1_dataLink[6].sName2:='N/A';
a1_dataLink[7].sName2:='N/A';
a1_dataLink[8].sName2:='Sec';
a1_dataLink[9].sName2:='Sec';
a1_dataLink[10].sName2:='Sec';
a1_dataLink[11].sName2:='Sec';
a1_dataLink[12].sName2:='Sec';
a1_dataLink[13].sName2:='Sec';
a1_dataLink[14].sName2:='DegC';
a1_dataLink[15].sName2:='DegC';
a1_dataLink[16].sName2:='%';
a1_dataLink[17].sName2:='%';
a1_dataLink[18].sName2:='Hz';
a1_dataLink[19].sName2:='Hz';
a1_dataLink[20].sName2:='%';
a1_dataLink[21].sName2:='%';
a1_dataLink[22].sName2:='Hz';
a1_dataLink[23].sName2:='Hz';
a1_dataLink[24].sName2:='%';
a1_dataLink[25].sName2:='%';
a1_dataLink[26].sName2:='Hz';
a1_dataLink[27].sName2:='Hz';
a1_dataLink[28].sName2:='%';
a1_dataLink[29].sName2:='%';
a1_dataLink[30].sName2:='Hz';
a1_dataLink[31].sName2:='Hz';
a1_dataLink[32].sName2:='Kpa';
a1_dataLink[33].sName2:='Kpa';
a1_dataLink[34].sName2:='uS';
a1_dataLink[35].sName2:='uS';
a1_dataLink[36].sName2:='LPM';
a1_dataLink[37].sName2:='LPM';
a1_dataLink[38].sName2:='OHM';
a1_dataLink[39].sName2:='OHM';
a1_dataLink[40].sName2:='PH';
a1_dataLink[41].sName2:='PH';
a1_dataLink[42].sName2:='N/A';
a1_dataLink[43].sName2:='N/A';
a1_dataLink[44].sName2:='Sec';
a1_dataLink[45].sName2:='Sec';


a1_dataLink[1].sName:='Station';
a1_dataLink[2].sName:='Station';
a1_dataLink[3].sName:='Sequences Recipe';
a1_dataLink[4].sName:='Sequences Recipe';
a1_dataLink[5].sName:='Sub Recipe';
a1_dataLink[6].sName:='Sub Recipe';
a1_dataLink[7].sName:='Minimum Time';
a1_dataLink[8].sName:='Minimum Time';
a1_dataLink[9].sName:='Maximum Time';
a1_dataLink[10].sName:='Maximum Time';
a1_dataLink[11].sName:='Effective Time';
a1_dataLink[12].sName:='Effective Time';
a1_dataLink[13].sName:='Temperature';
a1_dataLink[14].sName:='Temperature';
a1_dataLink[15].sName:='U/Sonic Bottom A Power';
a1_dataLink[16].sName:='U/Sonic Bottom A Power';
a1_dataLink[17].sName:='U/Sonic Bottom A Frequency';
a1_dataLink[18].sName:='U/Sonic Bottom A Frequency';
a1_dataLink[19].sName:='U/Sonic Bottom B Power';
a1_dataLink[20].sName:='U/Sonic Bottom B Power';
a1_dataLink[21].sName:='U/Sonic Bottom B Frequency';
a1_dataLink[22].sName:='U/Sonic Bottom B Frequency';
a1_dataLink[23].sName:='U/Sonic Side A Power SV';
a1_dataLink[24].sName:='U/Sonic Side A Power PV';
a1_dataLink[25].sName:='U/Sonic Side A Frequency';
a1_dataLink[26].sName:='U/Sonic Side A Frequency';
a1_dataLink[27].sName:='U/Sonic Side B Power';
a1_dataLink[28].sName:='U/Sonic Side B Power';
a1_dataLink[29].sName:='U/Sonic Side B Frequency';
a1_dataLink[30].sName:='U/Sonic Side B Frequency';
a1_dataLink[31].sName:='Vacuum SV';
a1_dataLink[32].sName:='Vacuum PV';
a1_dataLink[33].sName:='Conductivity';
a1_dataLink[34].sName:='Conductivity';
a1_dataLink[35].sName:='Pump Flow';
a1_dataLink[36].sName:='Pump Flow';
a1_dataLink[37].sName:='Resistivity';
a1_dataLink[38].sName:='Resistivity';
a1_dataLink[39].sName:='PH PV';
a1_dataLink[40].sName:='PH PV';
a1_dataLink[41].sName:='Quality';
a1_dataLink[42].sName:='Quality';
a1_dataLink[43].sName:='Actual Time';
a1_dataLink[44].sName:='Actual Time';


a1_dataLink[1].sValue:='N/A';(*Station*)
a1_dataLink[2].sValue:='1-US Cleaning';(*Station*)
a1_dataLink[3].sValue:='N/A';(*Sequences Recipe*)
a1_dataLink[4].sValue:=DSHmiStationDisplayInfo[1].sStationSequenceRecipeDescription;(*Sequences Recipe*)
a1_dataLink[5].sValue:='N/A';(*Sub Recipe*)
a1_dataLink[6].sValue:=DSHmiStationDisplayInfo[1].sStationSubDescription;(*Sub Recipe*)
a1_dataLink[7].sValue:=INT_TO_STRING(ARDsStnMinMaxEffTimeDisplay[1].iMinTime);(*Minimum Time*)
a1_dataLink[8].sValue:='N/A';(*Minimum Time*)
a1_dataLink[9].sValue:=INT_TO_STRING(ARDsStnMinMaxEffTimeDisplay[1].iMaxTime);(*Maximum Time*)
a1_dataLink[10].sValue:='N/A';(*Maximum Time*)
a1_dataLink[11].sValue:=INT_TO_STRING(ARDsStnMinMaxEffTimeDisplay[1].iEffTime);(*Effective Time*)
a1_dataLink[12].sValue:='N/A';(*Effective Time*)
a1_dataLink[13].sValue:=REAL_TO_STRING(ARrStnTempSV[1]);(*Temperature SV*)
a1_dataLink[14].sValue:=REAL_TO_STRING(ARrStnTempPV[1]);(*Temperature PV*)
a1_dataLink[15].sValue:=INT_TO_STRING(ARiStnManualUSBtmAsv[1]);(*U/Sonic Bottom A Power SV*)
a1_dataLink[16].sValue:=INT_TO_STRING(ARiStnUSBtmAPv[1]);(*U/Sonic Bottom A Power PV*)
a1_dataLink[17].sValue:='N/A';(*U/Sonic Bottom A Frequency SV*)
a1_dataLink[18].sValue:=INT_TO_STRING(DSWeberEnclosure[1].DSWeberGenerator[1].IN_iFreqSetPoint);(*U/Sonic Bottom A Frequency PV*)
a1_dataLink[19].sValue:=INT_TO_STRING(ARiStnManualUSBtmBsv[1]);(*U/Sonic Bottom B Power SV*)
a1_dataLink[20].sValue:=INT_TO_STRING(ARiStnUSBtmBPv[1]);(*U/Sonic Bottom B Power PV*)
a1_dataLink[21].sValue:='N/A';(*U/Sonic Bottom B Frequency SV*)
a1_dataLink[22].sValue:='N/A';(*U/Sonic Bottom B Frequency PV*)
a1_dataLink[23].sValue:='N/A';(*U/Sonic Side A Power SV*)
a1_dataLink[24].sValue:='N/A';(*U/Sonic Side A Power PV*)
a1_dataLink[25].sValue:='N/A';(*U/Sonic Side A Frequency SV*)
a1_dataLink[26].sValue:='N/A';(*U/Sonic Side A Frequency PV*)
a1_dataLink[27].sValue:='N/A';(*U/Sonic Side B Power SV*)
a1_dataLink[28].sValue:='N/A';(*U/Sonic Side B Power PV*)
a1_dataLink[29].sValue:='N/A';(*U/Sonic Side B Frequency SV*)
a1_dataLink[30].sValue:='N/A';(*U/Sonic Side B Frequency PV*)
a1_dataLink[31].sValue:='N/A';(*Vacuum SV*)
a1_dataLink[32].sValue:='N/A';(*Vacuum PV*)
a1_dataLink[33].sValue:='N/A';(*Conductivity SV*)
a1_dataLink[34].sValue:=REAL_TO_STRING(ARrStnConductivityPV[1]);(*Conductivity PV*)
a1_dataLink[35].sValue:='N/A';(*Pump Flow SV*)
a1_dataLink[36].sValue:=REAL_TO_STRING(ARrStnFilterPressurePV[1]);(*Pump Flow PV*)
a1_dataLink[37].sValue:='N/A';(*Resistivity SV*)
a1_dataLink[38].sValue:='N/A';(*Resistivity PV*)
a1_dataLink[39].sValue:='N/A';(*PH SV*)
a1_dataLink[40].sValue:='N/A'; (*PH PV*)
a1_dataLink[41].sValue:='N/A';(*Quality*)
a1_dataLink[42].sValue:=DSStnBasketInfo[1].sProductQuality;(*Quality*)
a1_dataLink[43].sValue:=INT_TO_STRING(ARDsStnSeqProcessCtrl[1].Out_iCurrentProcessTime);(*Actual Time*)
a1_dataLink[44].sValue:='N/A';(*Actual Time*)


(************************************************************************************************************************)

a2_dataLink[1].sName4:='';
a2_dataLink[2].sName4:='Operator';
a2_dataLink[3].sName4:='LD ID';
a2_dataLink[4].sName4:='ULD ID';
a2_dataLink[5].sName4:='Pro Recipe No';
a2_dataLink[6].sName4:='Pro Recipe Dscrp';
a2_dataLink[7].sName4:='LD No';


a2_dataLink[1].sName3:='';
a2_dataLink[2].sName3:=sUserName;
a2_dataLink[3].sName3:='1';
a2_dataLink[4].sName3:='1';
a2_dataLink[5].sName3:=INT_TO_STRING(DSStnBasketInfo[2].iProductRecipeNo);
a2_dataLink[6].sName3:=DSStnBasketInfo[2].sProgramDescription;
a2_dataLink[7].sName3:=INT_TO_STRING(iProgBatchTotal);


a2_dataLink[1].sName2:='';
a2_dataLink[2].sName2:='N/A';
a2_dataLink[3].sName2:='N/A';
a2_dataLink[4].sName2:='N/A';
a2_dataLink[5].sName2:='N/A';
a2_dataLink[6].sName2:='N/A';
a2_dataLink[7].sName2:='N/A';
a2_dataLink[8].sName2:='Sec';
a2_dataLink[9].sName2:='Sec';
a2_dataLink[10].sName2:='Sec';
a2_dataLink[11].sName2:='Sec';
a2_dataLink[12].sName2:='Sec';
a2_dataLink[13].sName2:='Sec';
a2_dataLink[14].sName2:='DegC';
a2_dataLink[15].sName2:='DegC';
a2_dataLink[16].sName2:='%';
a2_dataLink[17].sName2:='%';
a2_dataLink[18].sName2:='Hz';
a2_dataLink[19].sName2:='Hz';
a2_dataLink[20].sName2:='%';
a2_dataLink[21].sName2:='%';
a2_dataLink[22].sName2:='Hz';
a2_dataLink[23].sName2:='Hz';
a2_dataLink[24].sName2:='%';
a2_dataLink[25].sName2:='%';
a2_dataLink[26].sName2:='Hz';
a2_dataLink[27].sName2:='Hz';
a2_dataLink[28].sName2:='%';
a2_dataLink[29].sName2:='%';
a2_dataLink[30].sName2:='Hz';
a2_dataLink[31].sName2:='Hz';
a2_dataLink[32].sName2:='Kpa';
a2_dataLink[33].sName2:='Kpa';
a2_dataLink[34].sName2:='uS';
a2_dataLink[35].sName2:='uS';
a2_dataLink[36].sName2:='LPM';
a2_dataLink[37].sName2:='LPM';
a2_dataLink[38].sName2:='OHM';
a2_dataLink[39].sName2:='OHM';
a2_dataLink[40].sName2:='PH';
a2_dataLink[41].sName2:='PH';
a2_dataLink[42].sName2:='N/A';
a2_dataLink[43].sName2:='N/A';
a2_dataLink[44].sName2:='Sec';
a2_dataLink[45].sName2:='Sec';


a2_dataLink[1].sName:='Station';
a2_dataLink[2].sName:='Station';
a2_dataLink[3].sName:='Sequences Recipe';
a2_dataLink[4].sName:='Sequences Recipe';
a2_dataLink[5].sName:='Sub Recipe';
a2_dataLink[6].sName:='Sub Recipe';
a2_dataLink[7].sName:='Minimum Time';
a2_dataLink[8].sName:='Minimum Time';
a2_dataLink[9].sName:='Maximum Time';
a2_dataLink[10].sName:='Maximum Time';
a2_dataLink[11].sName:='Effective Time';
a2_dataLink[12].sName:='Effective Time';
a2_dataLink[13].sName:='Temperature';
a2_dataLink[14].sName:='Temperature';
a2_dataLink[15].sName:='U/Sonic Bottom A Power';
a2_dataLink[16].sName:='U/Sonic Bottom A Power';
a2_dataLink[17].sName:='U/Sonic Bottom A Frequency';
a2_dataLink[18].sName:='U/Sonic Bottom A Frequency';
a2_dataLink[19].sName:='U/Sonic Bottom B Power';
a2_dataLink[20].sName:='U/Sonic Bottom B Power';
a2_dataLink[21].sName:='U/Sonic Bottom B Frequency';
a2_dataLink[22].sName:='U/Sonic Bottom B Frequency';
a2_dataLink[23].sName:='U/Sonic Side A Power SV';
a2_dataLink[24].sName:='U/Sonic Side A Power PV';
a2_dataLink[25].sName:='U/Sonic Side A Frequency';
a2_dataLink[26].sName:='U/Sonic Side A Frequency';
a2_dataLink[27].sName:='U/Sonic Side B Power';
a2_dataLink[28].sName:='U/Sonic Side B Power';
a2_dataLink[29].sName:='U/Sonic Side B Frequency';
a2_dataLink[30].sName:='U/Sonic Side B Frequency';
a2_dataLink[31].sName:='Vacuum SV';
a2_dataLink[32].sName:='Vacuum PV';
a2_dataLink[33].sName:='Conductivity';
a2_dataLink[34].sName:='Conductivity';
a2_dataLink[35].sName:='Pump Flow';
a2_dataLink[36].sName:='Pump Flow';
a2_dataLink[37].sName:='Resistivity';
a2_dataLink[38].sName:='Resistivity';
a2_dataLink[39].sName:='PH PV';
a2_dataLink[40].sName:='PH PV';
a2_dataLink[41].sName:='Quality';
a2_dataLink[42].sName:='Quality';
a2_dataLink[43].sName:='Actual Time';
a2_dataLink[44].sName:='Actual Time';


a2_dataLink[1].sValue:='N/A';(*Station*)
a2_dataLink[2].sValue:='2-US Cleaning';(*Station*)
a2_dataLink[3].sValue:='N/A';(*Sequences Recipe*)
a2_dataLink[4].sValue:=DSHmiStationDisplayInfo[2].sStationSequenceRecipeDescription;(*Sequences Recipe*)
a2_dataLink[5].sValue:='N/A';(*Sub Recipe*)
a2_dataLink[6].sValue:=DSHmiStationDisplayInfo[2].sStationSubDescription;(*Sub Recipe*)
a2_dataLink[7].sValue:=INT_TO_STRING(ARDsStnMinMaxEffTimeDisplay[2].iMinTime);(*Minimum Time*)
a2_dataLink[8].sValue:='N/A';(*Minimum Time*)
a2_dataLink[9].sValue:=INT_TO_STRING(ARDsStnMinMaxEffTimeDisplay[2].iMaxTime);(*Maximum Time*)
a2_dataLink[10].sValue:='N/A';(*Maximum Time*)
a2_dataLink[11].sValue:=INT_TO_STRING(ARDsStnMinMaxEffTimeDisplay[2].iEffTime);(*Effective Time*)
a2_dataLink[12].sValue:='N/A';(*Effective Time*)
a2_dataLink[13].sValue:=REAL_TO_STRING(ARrStnTempSV[2]);(*Temperature SV*)
a2_dataLink[14].sValue:=REAL_TO_STRING(ARrStnTempPV[2]);(*Temperature PV*)
a2_dataLink[15].sValue:=INT_TO_STRING(ARiStnManualUSBtmAsv[2]);(*U/Sonic Bottom A Power SV*)
a2_dataLink[16].sValue:=INT_TO_STRING(ARiStnUSBtmAPv[2]);(*U/Sonic Bottom A Power PV*)
a2_dataLink[17].sValue:='N/A';(*U/Sonic Bottom A Frequency SV*)
a2_dataLink[18].sValue:=INT_TO_STRING(DSWeberEnclosure[1].DSWeberGenerator[2].IN_iFreqSetPoint);(*U/Sonic Bottom A Frequency PV*)
a2_dataLink[19].sValue:=INT_TO_STRING(ARiStnManualUSBtmBsv[2]);(*U/Sonic Bottom B Power SV*)
a2_dataLink[20].sValue:=INT_TO_STRING(ARiStnUSBtmBPv[2]);(*U/Sonic Bottom B Power PV*)
a2_dataLink[21].sValue:='N/A';(*U/Sonic Bottom B Frequency SV*)
a2_dataLink[22].sValue:='N/A';(*U/Sonic Bottom B Frequency PV*)
a2_dataLink[23].sValue:='N/A';(*U/Sonic Side A Power SV*)
a2_dataLink[24].sValue:='N/A';(*U/Sonic Side A Power PV*)
a2_dataLink[25].sValue:='N/A';(*U/Sonic Side A Frequency SV*)
a2_dataLink[26].sValue:='N/A';(*U/Sonic Side A Frequency PV*)
a2_dataLink[27].sValue:='N/A';(*U/Sonic Side B Power SV*)
a2_dataLink[28].sValue:='N/A';(*U/Sonic Side B Power PV*)
a2_dataLink[29].sValue:='N/A';(*U/Sonic Side B Frequency SV*)
a2_dataLink[30].sValue:='N/A';(*U/Sonic Side B Frequency PV*)
a2_dataLink[31].sValue:='N/A';(*Vacuum SV*)
a2_dataLink[32].sValue:='N/A';(*Vacuum PV*)
a2_dataLink[33].sValue:='N/A';(*Conductivity SV*)
a2_dataLink[34].sValue:=REAL_TO_STRING(ARrStnConductivityPV[2]);(*Conductivity PV*)
a2_dataLink[35].sValue:='N/A';(*Pump Flow SV*)
a2_dataLink[36].sValue:=REAL_TO_STRING(ARrStnFilterPressurePV[2]);(*Pump Flow PV*)
a2_dataLink[37].sValue:='N/A';(*Resistivity SV*)
a2_dataLink[38].sValue:='N/A';(*Resistivity PV*)
a2_dataLink[39].sValue:='N/A';(*PH SV*)
a2_dataLink[40].sValue:='N/A'; (*PH PV*)
a2_dataLink[41].sValue:='N/A';(*Quality*)
a2_dataLink[42].sValue:=DSStnBasketInfo[2].sProductQuality;(*Quality*)
a2_dataLink[43].sValue:=INT_TO_STRING(ARDsStnSeqProcessCtrl[2].Out_iCurrentProcessTime);(*Actual Time*)
a2_dataLink[44].sValue:='N/A';(*Actual Time*)

(************************************************************************************************************************)

a3_dataLink[1].sName4:='';
a3_dataLink[2].sName4:='Operator';
a3_dataLink[3].sName4:='LD ID';
a3_dataLink[4].sName4:='ULD ID';
a3_dataLink[5].sName4:='Pro Recipe No';
a3_dataLink[6].sName4:='Pro Recipe Dscrp';
a3_dataLink[7].sName4:='LD No';


a3_dataLink[1].sName3:='';
a3_dataLink[2].sName3:=sUserName;
a3_dataLink[3].sName3:='1';
a3_dataLink[4].sName3:='1';
a3_dataLink[5].sName3:=INT_TO_STRING(DSStnBasketInfo[3].iProductRecipeNo);
a3_dataLink[6].sName3:=DSStnBasketInfo[3].sProgramDescription;
a3_dataLink[7].sName3:=INT_TO_STRING(iProgBatchTotal);


a3_dataLink[1].sName2:='';
a3_dataLink[2].sName2:='N/A';
a3_dataLink[3].sName2:='N/A';
a3_dataLink[4].sName2:='N/A';
a3_dataLink[5].sName2:='N/A';
a3_dataLink[6].sName2:='N/A';
a3_dataLink[7].sName2:='N/A';
a3_dataLink[8].sName2:='Sec';
a3_dataLink[9].sName2:='Sec';
a3_dataLink[10].sName2:='Sec';
a3_dataLink[11].sName2:='Sec';
a3_dataLink[12].sName2:='Sec';
a3_dataLink[13].sName2:='Sec';
a3_dataLink[14].sName2:='DegC';
a3_dataLink[15].sName2:='DegC';
a3_dataLink[16].sName2:='%';
a3_dataLink[17].sName2:='%';
a3_dataLink[18].sName2:='Hz';
a3_dataLink[19].sName2:='Hz';
a3_dataLink[20].sName2:='%';
a3_dataLink[21].sName2:='%';
a3_dataLink[22].sName2:='Hz';
a3_dataLink[23].sName2:='Hz';
a3_dataLink[24].sName2:='%';
a3_dataLink[25].sName2:='%';
a3_dataLink[26].sName2:='Hz';
a3_dataLink[27].sName2:='Hz';
a3_dataLink[28].sName2:='%';
a3_dataLink[29].sName2:='%';
a3_dataLink[30].sName2:='Hz';
a3_dataLink[31].sName2:='Hz';
a3_dataLink[32].sName2:='Kpa';
a3_dataLink[33].sName2:='Kpa';
a3_dataLink[34].sName2:='uS';
a3_dataLink[35].sName2:='uS';
a3_dataLink[36].sName2:='LPM';
a3_dataLink[37].sName2:='LPM';
a3_dataLink[38].sName2:='OHM';
a3_dataLink[39].sName2:='OHM';
a3_dataLink[40].sName2:='PH';
a3_dataLink[41].sName2:='PH';
a3_dataLink[42].sName2:='N/A';
a3_dataLink[43].sName2:='N/A';
a3_dataLink[44].sName2:='Sec';
a3_dataLink[45].sName2:='Sec';



a3_dataLink[1].sName:='Station';
a3_dataLink[2].sName:='Station';
a3_dataLink[3].sName:='Sequences Recipe';
a3_dataLink[4].sName:='Sequences Recipe';
a3_dataLink[5].sName:='Sub Recipe';
a3_dataLink[6].sName:='Sub Recipe';
a3_dataLink[7].sName:='Minimum Time';
a3_dataLink[8].sName:='Minimum Time';
a3_dataLink[9].sName:='Maximum Time';
a3_dataLink[10].sName:='Maximum Time';
a3_dataLink[11].sName:='Effective Time';
a3_dataLink[12].sName:='Effective Time';
a3_dataLink[13].sName:='Temperature';
a3_dataLink[14].sName:='Temperature';
a3_dataLink[15].sName:='U/Sonic Bottom A Power';
a3_dataLink[16].sName:='U/Sonic Bottom A Power';
a3_dataLink[17].sName:='U/Sonic Bottom A Frequency';
a3_dataLink[18].sName:='U/Sonic Bottom A Frequency';
a3_dataLink[19].sName:='U/Sonic Bottom B Power';
a3_dataLink[20].sName:='U/Sonic Bottom B Power';
a3_dataLink[21].sName:='U/Sonic Bottom B Frequency';
a3_dataLink[22].sName:='U/Sonic Bottom B Frequency';
a3_dataLink[23].sName:='U/Sonic Side A Power SV';
a3_dataLink[24].sName:='U/Sonic Side A Power PV';
a3_dataLink[25].sName:='U/Sonic Side A Frequency';
a3_dataLink[26].sName:='U/Sonic Side A Frequency';
a3_dataLink[27].sName:='U/Sonic Side B Power';
a3_dataLink[28].sName:='U/Sonic Side B Power';
a3_dataLink[29].sName:='U/Sonic Side B Frequency';
a3_dataLink[30].sName:='U/Sonic Side B Frequency';
a3_dataLink[31].sName:='Vacuum SV';
a3_dataLink[32].sName:='Vacuum PV';
a3_dataLink[33].sName:='Conductivity';
a3_dataLink[34].sName:='Conductivity';
a3_dataLink[35].sName:='Pump Flow';
a3_dataLink[36].sName:='Pump Flow';
a3_dataLink[37].sName:='Resistivity';
a3_dataLink[38].sName:='Resistivity';
a3_dataLink[39].sName:='PH PV';
a3_dataLink[40].sName:='PH PV';
a3_dataLink[41].sName:='Quality';
a3_dataLink[42].sName:='Quality';
a3_dataLink[43].sName:='Actual Time';
a3_dataLink[44].sName:='Actual Time';


a3_dataLink[1].sValue:='N/A';(*Station*)
a3_dataLink[2].sValue:='3-US Cleaning';(*Station*)
a3_dataLink[3].sValue:='N/A';(*Sequences Recipe*)
a3_dataLink[4].sValue:=DSHmiStationDisplayInfo[3].sStationSequenceRecipeDescription;(*Sequences Recipe*)
a3_dataLink[5].sValue:='N/A';(*Sub Recipe*)
a3_dataLink[6].sValue:=DSHmiStationDisplayInfo[3].sStationSubDescription;(*Sub Recipe*)
a3_dataLink[7].sValue:=INT_TO_STRING(ARDsStnMinMaxEffTimeDisplay[3].iMinTime);(*Minimum Time*)
a3_dataLink[8].sValue:='N/A';(*Minimum Time*)
a3_dataLink[9].sValue:=INT_TO_STRING(ARDsStnMinMaxEffTimeDisplay[3].iMaxTime);(*Maximum Time*)
a3_dataLink[10].sValue:='N/A';(*Maximum Time*)
a3_dataLink[11].sValue:=INT_TO_STRING(ARDsStnMinMaxEffTimeDisplay[3].iEffTime);(*Effective Time*)
a3_dataLink[12].sValue:='N/A';(*Effective Time*)
a3_dataLink[13].sValue:=REAL_TO_STRING(ARrStnTempSV[3]);(*Temperature SV*)
a3_dataLink[14].sValue:=REAL_TO_STRING(ARrStnTempPV[3]);(*Temperature PV*)
a3_dataLink[15].sValue:=INT_TO_STRING(ARiStnManualUSBtmAsv[3]);(*U/Sonic Bottom A Power SV*)
a3_dataLink[16].sValue:=INT_TO_STRING(ARiStnUSBtmAPv[3]);(*U/Sonic Bottom A Power PV*)
a3_dataLink[17].sValue:='N/A';(*U/Sonic Bottom A Frequency SV*)
a3_dataLink[18].sValue:=INT_TO_STRING(DSWeberEnclosure[1].DSWeberGenerator[3].IN_iFreqSetPoint);(*U/Sonic Bottom A Frequency PV*)
a3_dataLink[19].sValue:=INT_TO_STRING(ARiStnManualUSBtmBsv[3]);(*U/Sonic Bottom B Power SV*)
a3_dataLink[20].sValue:=INT_TO_STRING(ARiStnUSBtmBPv[3]);(*U/Sonic Bottom B Power PV*)
a3_dataLink[21].sValue:='N/A';(*U/Sonic Bottom B Frequency SV*)
a3_dataLink[22].sValue:='N/A';(*U/Sonic Bottom B Frequency PV*)
a3_dataLink[23].sValue:='N/A';(*U/Sonic Side A Power SV*)
a3_dataLink[24].sValue:='N/A';(*U/Sonic Side A Power PV*)
a3_dataLink[25].sValue:='N/A';(*U/Sonic Side A Frequency SV*)
a3_dataLink[26].sValue:='N/A';(*U/Sonic Side A Frequency PV*)
a3_dataLink[27].sValue:='N/A';(*U/Sonic Side B Power SV*)
a3_dataLink[28].sValue:='N/A';(*U/Sonic Side B Power PV*)
a3_dataLink[29].sValue:='N/A';(*U/Sonic Side B Frequency SV*)
a3_dataLink[30].sValue:='N/A';(*U/Sonic Side B Frequency PV*)
a3_dataLink[31].sValue:='N/A';(*Vacuum SV*)
a3_dataLink[32].sValue:='N/A';(*Vacuum PV*)
a3_dataLink[33].sValue:='N/A';(*Conductivity SV*)
a3_dataLink[34].sValue:=REAL_TO_STRING(ARrStnConductivityPV[3]);(*Conductivity PV*)
a3_dataLink[35].sValue:='N/A';(*Pump Flow SV*)
a3_dataLink[36].sValue:=REAL_TO_STRING(ARrStnFilterPressurePV[3]);(*Pump Flow PV*)
a3_dataLink[37].sValue:='N/A';(*Resistivity SV*)
a3_dataLink[38].sValue:='N/A';(*Resistivity PV*)
a3_dataLink[39].sValue:='N/A';(*PH SV*)
a3_dataLink[40].sValue:='N/A'; (*PH PV*)
a3_dataLink[41].sValue:='N/A';(*Quality*)
a3_dataLink[42].sValue:=DSStnBasketInfo[3].sProductQuality;(*Quality*)
a3_dataLink[43].sValue:=INT_TO_STRING(ARDsStnSeqProcessCtrl[3].Out_iCurrentProcessTime);(*Actual Time*)
a3_dataLink[44].sValue:='N/A';(*Actual Time*)

(************************************************************************************************************************)

a4_dataLink[1].sName4:='';
a4_dataLink[2].sName4:='Operator';
a4_dataLink[3].sName4:='LD ID';
a4_dataLink[4].sName4:='ULD ID';
a4_dataLink[5].sName4:='Pro Recipe No';
a4_dataLink[6].sName4:='Pro Recipe Dscrp';
a4_dataLink[7].sName4:='LD No';


a4_dataLink[1].sName3:='';
a4_dataLink[2].sName3:=sUserName;
a4_dataLink[3].sName3:='1';
a4_dataLink[4].sName3:='1';
a4_dataLink[5].sName3:=INT_TO_STRING(DSStnBasketInfo[4].iProductRecipeNo);
a4_dataLink[6].sName3:=DSStnBasketInfo[4].sProgramDescription;
a4_dataLink[7].sName3:=INT_TO_STRING(iProgBatchTotal);


a4_dataLink[1].sName2:='';
a4_dataLink[2].sName2:='N/A';
a4_dataLink[3].sName2:='N/A';
a4_dataLink[4].sName2:='N/A';
a4_dataLink[5].sName2:='N/A';
a4_dataLink[6].sName2:='N/A';
a4_dataLink[7].sName2:='N/A';
a4_dataLink[8].sName2:='Sec';
a4_dataLink[9].sName2:='Sec';
a4_dataLink[10].sName2:='Sec';
a4_dataLink[11].sName2:='Sec';
a4_dataLink[12].sName2:='Sec';
a4_dataLink[13].sName2:='Sec';
a4_dataLink[14].sName2:='DegC';
a4_dataLink[15].sName2:='DegC';
a4_dataLink[16].sName2:='%';
a4_dataLink[17].sName2:='%';
a4_dataLink[18].sName2:='Hz';
a4_dataLink[19].sName2:='Hz';
a4_dataLink[20].sName2:='%';
a4_dataLink[21].sName2:='%';
a4_dataLink[22].sName2:='Hz';
a4_dataLink[23].sName2:='Hz';
a4_dataLink[24].sName2:='%';
a4_dataLink[25].sName2:='%';
a4_dataLink[26].sName2:='Hz';
a4_dataLink[27].sName2:='Hz';
a4_dataLink[28].sName2:='%';
a4_dataLink[29].sName2:='%';
a4_dataLink[30].sName2:='Hz';
a4_dataLink[31].sName2:='Hz';
a4_dataLink[32].sName2:='Kpa';
a4_dataLink[33].sName2:='Kpa';
a4_dataLink[34].sName2:='uS';
a4_dataLink[35].sName2:='uS';
a4_dataLink[36].sName2:='LPM';
a4_dataLink[37].sName2:='LPM';
a4_dataLink[38].sName2:='OHM';
a4_dataLink[39].sName2:='OHM';
a4_dataLink[40].sName2:='PH';
a4_dataLink[41].sName2:='PH';
a4_dataLink[42].sName2:='N/A';
a4_dataLink[43].sName2:='N/A';
a4_dataLink[44].sName2:='Sec';
a4_dataLink[45].sName2:='Sec';


a4_dataLink[1].sName:='Station';
a4_dataLink[2].sName:='Station';
a4_dataLink[3].sName:='Sequences Recipe';
a4_dataLink[4].sName:='Sequences Recipe';
a4_dataLink[5].sName:='Sub Recipe';
a4_dataLink[6].sName:='Sub Recipe';
a4_dataLink[7].sName:='Minimum Time';
a4_dataLink[8].sName:='Minimum Time';
a4_dataLink[9].sName:='Maximum Time';
a4_dataLink[10].sName:='Maximum Time';
a4_dataLink[11].sName:='Effective Time';
a4_dataLink[12].sName:='Effective Time';
a4_dataLink[13].sName:='Temperature';
a4_dataLink[14].sName:='Temperature';
a4_dataLink[15].sName:='U/Sonic Bottom A Power';
a4_dataLink[16].sName:='U/Sonic Bottom A Power';
a4_dataLink[17].sName:='U/Sonic Bottom A Frequency';
a4_dataLink[18].sName:='U/Sonic Bottom A Frequency';
a4_dataLink[19].sName:='U/Sonic Bottom B Power';
a4_dataLink[20].sName:='U/Sonic Bottom B Power';
a4_dataLink[21].sName:='U/Sonic Bottom B Frequency';
a4_dataLink[22].sName:='U/Sonic Bottom B Frequency';
a4_dataLink[23].sName:='U/Sonic Side A Power SV';
a4_dataLink[24].sName:='U/Sonic Side A Power PV';
a4_dataLink[25].sName:='U/Sonic Side A Frequency';
a4_dataLink[26].sName:='U/Sonic Side A Frequency';
a4_dataLink[27].sName:='U/Sonic Side B Power';
a4_dataLink[28].sName:='U/Sonic Side B Power';
a4_dataLink[29].sName:='U/Sonic Side B Frequency';
a4_dataLink[30].sName:='U/Sonic Side B Frequency';
a4_dataLink[31].sName:='Vacuum SV';
a4_dataLink[32].sName:='Vacuum PV';
a4_dataLink[33].sName:='Conductivity';
a4_dataLink[34].sName:='Conductivity';
a4_dataLink[35].sName:='Pump Flow';
a4_dataLink[36].sName:='Pump Flow';
a4_dataLink[37].sName:='Resistivity';
a4_dataLink[38].sName:='Resistivity';
a4_dataLink[39].sName:='PH PV';
a4_dataLink[40].sName:='PH PV';
a4_dataLink[41].sName:='Quality';
a4_dataLink[42].sName:='Quality';
a4_dataLink[43].sName:='Actual Time';
a4_dataLink[44].sName:='Actual Time';


a4_dataLink[1].sValue:='N/A';(*Station*)
a4_dataLink[2].sValue:='4-Rinsing';(*Station*)
a4_dataLink[3].sValue:='N/A';(*Sequences Recipe*)
a4_dataLink[4].sValue:=DSHmiStationDisplayInfo[4].sStationSequenceRecipeDescription;(*Sequences Recipe*)
a4_dataLink[5].sValue:='N/A';(*Sub Recipe*)
a4_dataLink[6].sValue:=DSHmiStationDisplayInfo[4].sStationSubDescription;(*Sub Recipe*)
a4_dataLink[7].sValue:=INT_TO_STRING(ARDsStnMinMaxEffTimeDisplay[4].iMinTime);(*Minimum Time*)
a4_dataLink[8].sValue:='N/A';(*Minimum Time*)
a4_dataLink[9].sValue:=INT_TO_STRING(ARDsStnMinMaxEffTimeDisplay[4].iMaxTime);(*Maximum Time*)
a4_dataLink[10].sValue:='N/A';(*Maximum Time*)
a4_dataLink[11].sValue:=INT_TO_STRING(ARDsStnMinMaxEffTimeDisplay[4].iEffTime);(*Effective Time*)
a4_dataLink[12].sValue:='N/A';(*Effective Time*)
a4_dataLink[13].sValue:=REAL_TO_STRING(ARrStnTempSV[4]);(*Temperature SV*)
a4_dataLink[14].sValue:=REAL_TO_STRING(ARrStnTempPV[4]);(*Temperature PV*)
a4_dataLink[15].sValue:=INT_TO_STRING(ARiStnManualUSBtmAsv[4]);(*U/Sonic Bottom A Power SV*)
a4_dataLink[16].sValue:=INT_TO_STRING(ARiStnUSBtmAPv[4]);(*U/Sonic Bottom A Power PV*)
a4_dataLink[17].sValue:='N/A';(*U/Sonic Bottom A Frequency SV*)
a4_dataLink[18].sValue:='N/A';(*U/Sonic Bottom A Frequency PV*)
a4_dataLink[19].sValue:=INT_TO_STRING(ARiStnManualUSBtmBsv[4]);(*U/Sonic Bottom B Power SV*)
a4_dataLink[20].sValue:=INT_TO_STRING(ARiStnUSBtmBPv[4]);(*U/Sonic Bottom B Power PV*)
a4_dataLink[21].sValue:='N/A';(*U/Sonic Bottom B Frequency SV*)
a4_dataLink[22].sValue:='N/A';(*U/Sonic Bottom B Frequency PV*)
a4_dataLink[23].sValue:='N/A';(*U/Sonic Side A Power SV*)
a4_dataLink[24].sValue:='N/A';(*U/Sonic Side A Power PV*)
a4_dataLink[25].sValue:='N/A';(*U/Sonic Side A Frequency SV*)
a4_dataLink[26].sValue:='N/A';(*U/Sonic Side A Frequency PV*)
a4_dataLink[27].sValue:='N/A';(*U/Sonic Side B Power SV*)
a4_dataLink[28].sValue:='N/A';(*U/Sonic Side B Power PV*)
a4_dataLink[29].sValue:='N/A';(*U/Sonic Side B Frequency SV*)
a4_dataLink[30].sValue:='N/A';(*U/Sonic Side B Frequency PV*)
a4_dataLink[31].sValue:='N/A';(*Vacuum SV*)
a4_dataLink[32].sValue:='N/A';(*Vacuum PV*)
a4_dataLink[33].sValue:='N/A';(*Conductivity SV*)
a4_dataLink[34].sValue:=REAL_TO_STRING(ARrStnConductivityPV[4]);(*Conductivity PV*)
a4_dataLink[35].sValue:='N/A';(*Pump Flow SV*)
a4_dataLink[36].sValue:=REAL_TO_STRING(ARrStnFilterPressurePV[4]);(*Pump Flow PV*)
a4_dataLink[37].sValue:='N/A';(*Resistivity SV*)
a4_dataLink[38].sValue:='N/A';(*Resistivity PV*)
a4_dataLink[39].sValue:='N/A';(*PH SV*)
a4_dataLink[40].sValue:='N/A'; (*PH PV*)
a4_dataLink[41].sValue:='N/A';(*Quality*)
a4_dataLink[42].sValue:=DSStnBasketInfo[4].sProductQuality;(*Quality*)
a4_dataLink[43].sValue:=INT_TO_STRING(ARDsStnSeqProcessCtrl[4].Out_iCurrentProcessTime);(*Actual Time*)
a4_dataLink[44].sValue:='N/A';(*Actual Time*)

(************************************************************************************************************************)
a5_dataLink[1].sName4:='';
a5_dataLink[2].sName4:='Operator';
a5_dataLink[3].sName4:='LD ID';
a5_dataLink[4].sName4:='ULD ID';
a5_dataLink[5].sName4:='Pro Recipe No';
a5_dataLink[6].sName4:='Pro Recipe Dscrp';
a5_dataLink[7].sName4:='LD No';


a5_dataLink[1].sName3:='';
a5_dataLink[2].sName3:=sUserName;
a5_dataLink[3].sName3:='1';
a5_dataLink[4].sName3:='1';
a5_dataLink[5].sName3:=INT_TO_STRING(DSStnBasketInfo[5].iProductRecipeNo);
a5_dataLink[6].sName3:=DSStnBasketInfo[5].sProgramDescription;
a5_dataLink[7].sName3:=INT_TO_STRING(iProgBatchTotal);

a5_dataLink[1].sName2:='';
a5_dataLink[2].sName2:='N/A';
a5_dataLink[3].sName2:='N/A';
a5_dataLink[4].sName2:='N/A';
a5_dataLink[5].sName2:='N/A';
a5_dataLink[6].sName2:='N/A';
a5_dataLink[7].sName2:='N/A';
a5_dataLink[8].sName2:='Sec';
a5_dataLink[9].sName2:='Sec';
a5_dataLink[10].sName2:='Sec';
a5_dataLink[11].sName2:='Sec';
a5_dataLink[12].sName2:='Sec';
a5_dataLink[13].sName2:='Sec';
a5_dataLink[14].sName2:='DegC';
a5_dataLink[15].sName2:='DegC';
a5_dataLink[16].sName2:='%';
a5_dataLink[17].sName2:='%';
a5_dataLink[18].sName2:='Hz';
a5_dataLink[19].sName2:='Hz';
a5_dataLink[20].sName2:='%';
a5_dataLink[21].sName2:='%';
a5_dataLink[22].sName2:='Hz';
a5_dataLink[23].sName2:='Hz';
a5_dataLink[24].sName2:='%';
a5_dataLink[25].sName2:='%';
a5_dataLink[26].sName2:='Hz';
a5_dataLink[27].sName2:='Hz';
a5_dataLink[28].sName2:='%';
a5_dataLink[29].sName2:='%';
a5_dataLink[30].sName2:='Hz';
a5_dataLink[31].sName2:='Hz';
a5_dataLink[32].sName2:='Kpa';
a5_dataLink[33].sName2:='Kpa';
a5_dataLink[34].sName2:='uS';
a5_dataLink[35].sName2:='uS';
a5_dataLink[36].sName2:='LPM';
a5_dataLink[37].sName2:='LPM';
a5_dataLink[38].sName2:='OHM';
a5_dataLink[39].sName2:='OHM';
a5_dataLink[40].sName2:='PH';
a5_dataLink[41].sName2:='PH';
a5_dataLink[42].sName2:='N/A';
a5_dataLink[43].sName2:='N/A';
a5_dataLink[44].sName2:='Sec';
a5_dataLink[45].sName2:='Sec';



a5_dataLink[1].sName:='Station';
a5_dataLink[2].sName:='Station';
a5_dataLink[3].sName:='Sequences Recipe';
a5_dataLink[4].sName:='Sequences Recipe';
a5_dataLink[5].sName:='Sub Recipe';
a5_dataLink[6].sName:='Sub Recipe';
a5_dataLink[7].sName:='Minimum Time';
a5_dataLink[8].sName:='Minimum Time';
a5_dataLink[9].sName:='Maximum Time';
a5_dataLink[10].sName:='Maximum Time';
a5_dataLink[11].sName:='Effective Time';
a5_dataLink[12].sName:='Effective Time';
a5_dataLink[13].sName:='Temperature';
a5_dataLink[14].sName:='Temperature';
a5_dataLink[15].sName:='U/Sonic Bottom A Power';
a5_dataLink[16].sName:='U/Sonic Bottom A Power';
a5_dataLink[17].sName:='U/Sonic Bottom A Frequency';
a5_dataLink[18].sName:='U/Sonic Bottom A Frequency';
a5_dataLink[19].sName:='U/Sonic Bottom B Power';
a5_dataLink[20].sName:='U/Sonic Bottom B Power';
a5_dataLink[21].sName:='U/Sonic Bottom B Frequency';
a5_dataLink[22].sName:='U/Sonic Bottom B Frequency';
a5_dataLink[23].sName:='U/Sonic Side A Power SV';
a5_dataLink[24].sName:='U/Sonic Side A Power PV';
a5_dataLink[25].sName:='U/Sonic Side A Frequency';
a5_dataLink[26].sName:='U/Sonic Side A Frequency';
a5_dataLink[27].sName:='U/Sonic Side B Power';
a5_dataLink[28].sName:='U/Sonic Side B Power';
a5_dataLink[29].sName:='U/Sonic Side B Frequency';
a5_dataLink[30].sName:='U/Sonic Side B Frequency';
a5_dataLink[31].sName:='Vacuum SV';
a5_dataLink[32].sName:='Vacuum PV';
a5_dataLink[33].sName:='Conductivity';
a5_dataLink[34].sName:='Conductivity';
a5_dataLink[35].sName:='Pump Flow';
a5_dataLink[36].sName:='Pump Flow';
a5_dataLink[37].sName:='Resistivity';
a5_dataLink[38].sName:='Resistivity';
a5_dataLink[39].sName:='PH PV';
a5_dataLink[40].sName:='PH PV';
a5_dataLink[41].sName:='Quality';
a5_dataLink[42].sName:='Quality';
a5_dataLink[43].sName:='Actual Time';
a5_dataLink[44].sName:='Actual Time';


a5_dataLink[1].sValue:='N/A';(*Station*)
a5_dataLink[2].sValue:='5-US Cleaning';(*Station*)
a5_dataLink[3].sValue:='N/A';(*Sequences Recipe*)
a5_dataLink[4].sValue:=DSHmiStationDisplayInfo[5].sStationSequenceRecipeDescription;(*Sequences Recipe*)
a5_dataLink[5].sValue:='N/A';(*Sub Recipe*)
a5_dataLink[6].sValue:=DSHmiStationDisplayInfo[5].sStationSubDescription;(*Sub Recipe*)
a5_dataLink[7].sValue:=INT_TO_STRING(ARDsStnMinMaxEffTimeDisplay[5].iMinTime);(*Minimum Time*)
a5_dataLink[8].sValue:='N/A';(*Minimum Time*)
a5_dataLink[9].sValue:=INT_TO_STRING(ARDsStnMinMaxEffTimeDisplay[5].iMaxTime);(*Maximum Time*)
a5_dataLink[10].sValue:='N/A';(*Maximum Time*)
a5_dataLink[11].sValue:=INT_TO_STRING(ARDsStnMinMaxEffTimeDisplay[5].iEffTime);(*Effective Time*)
a5_dataLink[12].sValue:='N/A';(*Effective Time*)
a5_dataLink[13].sValue:=REAL_TO_STRING(ARrStnTempSV[5]);(*Temperature SV*)
a5_dataLink[14].sValue:=REAL_TO_STRING(ARrStnTempPV[5]);(*Temperature PV*)
a5_dataLink[15].sValue:=INT_TO_STRING(ARiStnManualUSBtmAsv[5]);(*U/Sonic Bottom A Power SV*)
a5_dataLink[16].sValue:=INT_TO_STRING(ARiStnUSBtmAPv[5]);(*U/Sonic Bottom A Power PV*)
a5_dataLink[17].sValue:='N/A';(*U/Sonic Bottom A Frequency SV*)
a5_dataLink[18].sValue:=INT_TO_STRING(DSWeberEnclosure[1].DSWeberGenerator[5].IN_iFreqSetPoint);(*U/Sonic Bottom A Frequency PV*)
a5_dataLink[19].sValue:=INT_TO_STRING(ARiStnManualUSBtmBsv[5]);(*U/Sonic Bottom B Power SV*)
a5_dataLink[20].sValue:=INT_TO_STRING(ARiStnUSBtmBPv[5]);(*U/Sonic Bottom B Power PV*)
a5_dataLink[21].sValue:='N/A';(*U/Sonic Bottom B Frequency SV*)
a5_dataLink[22].sValue:='N/A';(*U/Sonic Bottom B Frequency PV*)
a5_dataLink[23].sValue:='N/A';(*U/Sonic Side A Power SV*)
a5_dataLink[24].sValue:='N/A';(*U/Sonic Side A Power PV*)
a5_dataLink[25].sValue:='N/A';(*U/Sonic Side A Frequency SV*)
a5_dataLink[26].sValue:='N/A';(*U/Sonic Side A Frequency PV*)
a5_dataLink[27].sValue:='N/A';(*U/Sonic Side B Power SV*)
a5_dataLink[28].sValue:='N/A';(*U/Sonic Side B Power PV*)
a5_dataLink[29].sValue:='N/A';(*U/Sonic Side B Frequency SV*)
a5_dataLink[30].sValue:='N/A';(*U/Sonic Side B Frequency PV*)
a5_dataLink[31].sValue:='N/A';(*Vacuum SV*)
a5_dataLink[32].sValue:='N/A';(*Vacuum PV*)
a5_dataLink[33].sValue:='N/A';(*Conductivity SV*)
a5_dataLink[34].sValue:=REAL_TO_STRING(ARrStnConductivityPV[5]);(*Conductivity PV*)
a5_dataLink[35].sValue:='N/A';(*Pump Flow SV*)
a5_dataLink[36].sValue:=REAL_TO_STRING(ARrStnFilterPressurePV[5]);(*Pump Flow PV*)
a5_dataLink[37].sValue:='N/A';(*Resistivity SV*)
a5_dataLink[38].sValue:='N/A';(*Resistivity PV*)
a5_dataLink[39].sValue:='N/A';(*PH SV*)
a5_dataLink[40].sValue:=REAL_TO_STRING(ARrStnPhPV[5]); (*PH PV*)
a5_dataLink[41].sValue:='N/A';(*Quality*)
a5_dataLink[42].sValue:=DSStnBasketInfo[5].sProductQuality;(*Quality*)
a5_dataLink[43].sValue:=INT_TO_STRING(ARDsStnSeqProcessCtrl[5].Out_iCurrentProcessTime);(*Actual Time*)
a5_dataLink[44].sValue:='N/A';(*Actual Time*)

(************************************************************************************************************************)
a6_dataLink[1].sName4:='';
a6_dataLink[2].sName4:='Operator';
a6_dataLink[3].sName4:='LD ID';
a6_dataLink[4].sName4:='ULD ID';
a6_dataLink[5].sName4:='Pro Recipe No';
a6_dataLink[6].sName4:='Pro Recipe Dscrp';
a6_dataLink[7].sName4:='LD No';


a6_dataLink[1].sName3:='';
a6_dataLink[2].sName3:=sUserName;
a6_dataLink[3].sName3:='1';
a6_dataLink[4].sName3:='1';
a6_dataLink[5].sName3:=INT_TO_STRING(DSStnBasketInfo[6].iProductRecipeNo);
a6_dataLink[6].sName3:=DSStnBasketInfo[6].sProgramDescription;
a6_dataLink[7].sName3:=INT_TO_STRING(iProgBatchTotal);

a6_dataLink[1].sName2:='';
a6_dataLink[2].sName2:='N/A';
a6_dataLink[3].sName2:='N/A';
a6_dataLink[4].sName2:='N/A';
a6_dataLink[5].sName2:='N/A';
a6_dataLink[6].sName2:='N/A';
a6_dataLink[7].sName2:='N/A';
a6_dataLink[8].sName2:='Sec';
a6_dataLink[9].sName2:='Sec';
a6_dataLink[10].sName2:='Sec';
a6_dataLink[11].sName2:='Sec';
a6_dataLink[12].sName2:='Sec';
a6_dataLink[13].sName2:='Sec';
a6_dataLink[14].sName2:='DegC';
a6_dataLink[15].sName2:='DegC';
a6_dataLink[16].sName2:='%';
a6_dataLink[17].sName2:='%';
a6_dataLink[18].sName2:='Hz';
a6_dataLink[19].sName2:='Hz';
a6_dataLink[20].sName2:='%';
a6_dataLink[21].sName2:='%';
a6_dataLink[22].sName2:='Hz';
a6_dataLink[23].sName2:='Hz';
a6_dataLink[24].sName2:='%';
a6_dataLink[25].sName2:='%';
a6_dataLink[26].sName2:='Hz';
a6_dataLink[27].sName2:='Hz';
a6_dataLink[28].sName2:='%';
a6_dataLink[29].sName2:='%';
a6_dataLink[30].sName2:='Hz';
a6_dataLink[31].sName2:='Hz';
a6_dataLink[32].sName2:='Kpa';
a6_dataLink[33].sName2:='Kpa';
a6_dataLink[34].sName2:='uS';
a6_dataLink[35].sName2:='uS';
a6_dataLink[36].sName2:='LPM';
a6_dataLink[37].sName2:='LPM';
a6_dataLink[38].sName2:='OHM';
a6_dataLink[39].sName2:='OHM';
a6_dataLink[40].sName2:='PH';
a6_dataLink[41].sName2:='PH';
a6_dataLink[42].sName2:='N/A';
a6_dataLink[43].sName2:='N/A';
a6_dataLink[44].sName2:='Sec';
a6_dataLink[45].sName2:='Sec';



a6_dataLink[1].sName:='Station';
a6_dataLink[2].sName:='Station';
a6_dataLink[3].sName:='Sequences Recipe';
a6_dataLink[4].sName:='Sequences Recipe';
a6_dataLink[5].sName:='Sub Recipe';
a6_dataLink[6].sName:='Sub Recipe';
a6_dataLink[7].sName:='Minimum Time';
a6_dataLink[8].sName:='Minimum Time';
a6_dataLink[9].sName:='Maximum Time';
a6_dataLink[10].sName:='Maximum Time';
a6_dataLink[11].sName:='Effective Time';
a6_dataLink[12].sName:='Effective Time';
a6_dataLink[13].sName:='Temperature';
a6_dataLink[14].sName:='Temperature';
a6_dataLink[15].sName:='U/Sonic Bottom A Power';
a6_dataLink[16].sName:='U/Sonic Bottom A Power';
a6_dataLink[17].sName:='U/Sonic Bottom A Frequency';
a6_dataLink[18].sName:='U/Sonic Bottom A Frequency';
a6_dataLink[19].sName:='U/Sonic Bottom B Power';
a6_dataLink[20].sName:='U/Sonic Bottom B Power';
a6_dataLink[21].sName:='U/Sonic Bottom B Frequency';
a6_dataLink[22].sName:='U/Sonic Bottom B Frequency';
a6_dataLink[23].sName:='U/Sonic Side A Power SV';
a6_dataLink[24].sName:='U/Sonic Side A Power PV';
a6_dataLink[25].sName:='U/Sonic Side A Frequency';
a6_dataLink[26].sName:='U/Sonic Side A Frequency';
a6_dataLink[27].sName:='U/Sonic Side B Power';
a6_dataLink[28].sName:='U/Sonic Side B Power';
a6_dataLink[29].sName:='U/Sonic Side B Frequency';
a6_dataLink[30].sName:='U/Sonic Side B Frequency';
a6_dataLink[31].sName:='Vacuum SV';
a6_dataLink[32].sName:='Vacuum PV';
a6_dataLink[33].sName:='Conductivity';
a6_dataLink[34].sName:='Conductivity';
a6_dataLink[35].sName:='Pump Flow';
a6_dataLink[36].sName:='Pump Flow';
a6_dataLink[37].sName:='Resistivity';
a6_dataLink[38].sName:='Resistivity';
a6_dataLink[39].sName:='PH PV';
a6_dataLink[40].sName:='PH PV';
a6_dataLink[41].sName:='Quality';
a6_dataLink[42].sName:='Quality';
a6_dataLink[43].sName:='Actual Time';
a6_dataLink[44].sName:='Actual Time';


a6_dataLink[1].sValue:='N/A';(*Station*)
a6_dataLink[2].sValue:='6-Rinsing';(*Station*)
a6_dataLink[3].sValue:='N/A';(*Sequences Recipe*)
a6_dataLink[4].sValue:=DSHmiStationDisplayInfo[6].sStationSequenceRecipeDescription;(*Sequences Recipe*)
a6_dataLink[5].sValue:='N/A';(*Sub Recipe*)
a6_dataLink[6].sValue:=DSHmiStationDisplayInfo[6].sStationSubDescription;(*Sub Recipe*)
a6_dataLink[7].sValue:=INT_TO_STRING(ARDsStnMinMaxEffTimeDisplay[6].iMinTime);(*Minimum Time*)
a6_dataLink[8].sValue:='N/A';(*Minimum Time*)
a6_dataLink[9].sValue:=INT_TO_STRING(ARDsStnMinMaxEffTimeDisplay[6].iMaxTime);(*Maximum Time*)
a6_dataLink[10].sValue:='N/A';(*Maximum Time*)
a6_dataLink[11].sValue:=INT_TO_STRING(ARDsStnMinMaxEffTimeDisplay[6].iEffTime);(*Effective Time*)
a6_dataLink[12].sValue:='N/A';(*Effective Time*)
a6_dataLink[13].sValue:=REAL_TO_STRING(ARrStnTempSV[6]);(*Temperature SV*)
a6_dataLink[14].sValue:=REAL_TO_STRING(ARrStnTempPV[6]);(*Temperature PV*)
a6_dataLink[15].sValue:=INT_TO_STRING(ARiStnManualUSBtmAsv[6]);(*U/Sonic Bottom A Power SV*)
a6_dataLink[16].sValue:=INT_TO_STRING(ARiStnUSBtmAPv[6]);(*U/Sonic Bottom A Power PV*)
a6_dataLink[17].sValue:='N/A';(*U/Sonic Bottom A Frequency SV*)
a6_dataLink[18].sValue:='N/A';(*U/Sonic Bottom A Frequency PV*)
a6_dataLink[19].sValue:=INT_TO_STRING(ARiStnManualUSBtmBsv[6]);(*U/Sonic Bottom B Power SV*)
a6_dataLink[20].sValue:=INT_TO_STRING(ARiStnUSBtmBPv[6]);(*U/Sonic Bottom B Power PV*)
a6_dataLink[21].sValue:='N/A';(*U/Sonic Bottom B Frequency SV*)
a6_dataLink[22].sValue:='N/A';(*U/Sonic Bottom B Frequency PV*)
a6_dataLink[23].sValue:='N/A';(*U/Sonic Side A Power SV*)
a6_dataLink[24].sValue:='N/A';(*U/Sonic Side A Power PV*)
a6_dataLink[25].sValue:='N/A';(*U/Sonic Side A Frequency SV*)
a6_dataLink[26].sValue:='N/A';(*U/Sonic Side A Frequency PV*)
a6_dataLink[27].sValue:='N/A';(*U/Sonic Side B Power SV*)
a6_dataLink[28].sValue:='N/A';(*U/Sonic Side B Power PV*)
a6_dataLink[29].sValue:='N/A';(*U/Sonic Side B Frequency SV*)
a6_dataLink[30].sValue:='N/A';(*U/Sonic Side B Frequency PV*)
a6_dataLink[31].sValue:='N/A';(*Vacuum SV*)
a6_dataLink[32].sValue:='N/A';(*Vacuum PV*)
a6_dataLink[33].sValue:='N/A';(*Conductivity SV*)
a6_dataLink[34].sValue:=REAL_TO_STRING(ARrStnConductivityPV[6]);(*Conductivity PV*)
a6_dataLink[35].sValue:='N/A';(*Pump Flow SV*)
a6_dataLink[36].sValue:=REAL_TO_STRING(ARrStnFilterPressurePV[6]);(*Pump Flow PV*)
a6_dataLink[37].sValue:='N/A';(*Resistivity SV*)
a6_dataLink[38].sValue:='N/A';(*Resistivity PV*)
a6_dataLink[39].sValue:='N/A';(*PH SV*)
a6_dataLink[40].sValue:='N/A'; (*PH PV*)
a6_dataLink[41].sValue:='N/A';(*Quality*)
a6_dataLink[42].sValue:=DSStnBasketInfo[6].sProductQuality;(*Quality*)
a6_dataLink[43].sValue:=INT_TO_STRING(ARDsStnSeqProcessCtrl[6].Out_iCurrentProcessTime);(*Actual Time*)
a6_dataLink[44].sValue:='N/A';(*Actual Time*)

(************************************************************************************************************************)
a7_dataLink[1].sName4:='';
a7_dataLink[2].sName4:='Operator';
a7_dataLink[3].sName4:='LD ID';
a7_dataLink[4].sName4:='ULD ID';
a7_dataLink[5].sName4:='Pro Recipe No';
a7_dataLink[6].sName4:='Pro Recipe Dscrp';
a7_dataLink[7].sName4:='LD No';


a7_dataLink[1].sName3:='';
a7_dataLink[2].sName3:=sUserName;
a7_dataLink[3].sName3:='1';
a7_dataLink[4].sName3:='1';
a7_dataLink[5].sName3:=INT_TO_STRING(DSStnBasketInfo[7].iProductRecipeNo);
a7_dataLink[6].sName3:=DSStnBasketInfo[7].sProgramDescription;
a7_dataLink[7].sName3:=INT_TO_STRING(iProgBatchTotal);

a7_dataLink[1].sName2:='';
a7_dataLink[2].sName2:='N/A';
a7_dataLink[3].sName2:='N/A';
a7_dataLink[4].sName2:='N/A';
a7_dataLink[5].sName2:='N/A';
a7_dataLink[6].sName2:='N/A';
a7_dataLink[7].sName2:='N/A';
a7_dataLink[8].sName2:='Sec';
a7_dataLink[9].sName2:='Sec';
a7_dataLink[10].sName2:='Sec';
a7_dataLink[11].sName2:='Sec';
a7_dataLink[12].sName2:='Sec';
a7_dataLink[13].sName2:='Sec';
a7_dataLink[14].sName2:='DegC';
a7_dataLink[15].sName2:='DegC';
a7_dataLink[16].sName2:='%';
a7_dataLink[17].sName2:='%';
a7_dataLink[18].sName2:='Hz';
a7_dataLink[19].sName2:='Hz';
a7_dataLink[20].sName2:='%';
a7_dataLink[21].sName2:='%';
a7_dataLink[22].sName2:='Hz';
a7_dataLink[23].sName2:='Hz';
a7_dataLink[24].sName2:='%';
a7_dataLink[25].sName2:='%';
a7_dataLink[26].sName2:='Hz';
a7_dataLink[27].sName2:='Hz';
a7_dataLink[28].sName2:='%';
a7_dataLink[29].sName2:='%';
a7_dataLink[30].sName2:='Hz';
a7_dataLink[31].sName2:='Hz';
a7_dataLink[32].sName2:='Kpa';
a7_dataLink[33].sName2:='Kpa';
a7_dataLink[34].sName2:='uS';
a7_dataLink[35].sName2:='uS';
a7_dataLink[36].sName2:='LPM';
a7_dataLink[37].sName2:='LPM';
a7_dataLink[38].sName2:='OHM';
a7_dataLink[39].sName2:='OHM';
a7_dataLink[40].sName2:='PH';
a7_dataLink[41].sName2:='PH';
a7_dataLink[42].sName2:='N/A';
a7_dataLink[43].sName2:='N/A';
a7_dataLink[44].sName2:='Sec';
a7_dataLink[45].sName2:='Sec';



a7_dataLink[1].sName:='Station';
a7_dataLink[2].sName:='Station';
a7_dataLink[3].sName:='Sequences Recipe';
a7_dataLink[4].sName:='Sequences Recipe';
a7_dataLink[5].sName:='Sub Recipe';
a7_dataLink[6].sName:='Sub Recipe';
a7_dataLink[7].sName:='Minimum Time';
a7_dataLink[8].sName:='Minimum Time';
a7_dataLink[9].sName:='Maximum Time';
a7_dataLink[10].sName:='Maximum Time';
a7_dataLink[11].sName:='Effective Time';
a7_dataLink[12].sName:='Effective Time';
a7_dataLink[13].sName:='Temperature';
a7_dataLink[14].sName:='Temperature';
a7_dataLink[15].sName:='U/Sonic Bottom A Power';
a7_dataLink[16].sName:='U/Sonic Bottom A Power';
a7_dataLink[17].sName:='U/Sonic Bottom A Frequency';
a7_dataLink[18].sName:='U/Sonic Bottom A Frequency';
a7_dataLink[19].sName:='U/Sonic Bottom B Power';
a7_dataLink[20].sName:='U/Sonic Bottom B Power';
a7_dataLink[21].sName:='U/Sonic Bottom B Frequency';
a7_dataLink[22].sName:='U/Sonic Bottom B Frequency';
a7_dataLink[23].sName:='U/Sonic Side A Power SV';
a7_dataLink[24].sName:='U/Sonic Side A Power PV';
a7_dataLink[25].sName:='U/Sonic Side A frequency';
a7_dataLink[26].sName:='U/Sonic Side A frequency';
a7_dataLink[27].sName:='U/Sonic Side B Power';
a7_dataLink[28].sName:='U/Sonic Side B Power';
a7_dataLink[29].sName:='U/Sonic Side B Frequency';
a7_dataLink[30].sName:='U/Sonic Side B Frequency';
a7_dataLink[31].sName:='Vacuum SV';
a7_dataLink[32].sName:='Vacuum PV';
a7_dataLink[33].sName:='Conductivity';
a7_dataLink[34].sName:='Conductivity';
a7_dataLink[35].sName:='Pump Flow';
a7_dataLink[36].sName:='Pump Flow';
a7_dataLink[37].sName:='Resistivity';
a7_dataLink[38].sName:='Resistivity';
a7_dataLink[39].sName:='PH PV';
a7_dataLink[40].sName:='PH PV';
a7_dataLink[41].sName:='Quality';
a7_dataLink[42].sName:='Quality';
a7_dataLink[43].sName:='Actual Time';
a7_dataLink[44].sName:='Actual Time';


a7_dataLink[1].sValue:='N/A';(*Station*)
a7_dataLink[2].sValue:='7-US Rinsing DI';(*Station*)
a7_dataLink[3].sValue:='N/A';(*Sequences Recipe*)
a7_dataLink[4].sValue:=DSHmiStationDisplayInfo[7].sStationSequenceRecipeDescription;(*Sequences Recipe*)
a7_dataLink[5].sValue:='N/A';(*Sub Recipe*)
a7_dataLink[6].sValue:=DSHmiStationDisplayInfo[7].sStationSubDescription;(*Sub Recipe*)
a7_dataLink[7].sValue:=INT_TO_STRING(ARDsStnMinMaxEffTimeDisplay[7].iMinTime);(*Minimum Time*)
a7_dataLink[8].sValue:='N/A';(*Minimum Time*)
a7_dataLink[9].sValue:=INT_TO_STRING(ARDsStnMinMaxEffTimeDisplay[7].iMaxTime);(*Maximum Time*)
a7_dataLink[10].sValue:='N/A';(*Maximum Time*)
a7_dataLink[11].sValue:=INT_TO_STRING(ARDsStnMinMaxEffTimeDisplay[7].iEffTime);(*Effective Time*)
a7_dataLink[12].sValue:='N/A';(*Effective Time*)
a7_dataLink[13].sValue:=REAL_TO_STRING(ARrStnTempSV[7]);(*Temperature SV*)
a7_dataLink[14].sValue:=REAL_TO_STRING(ARrStnTempPV[7]);(*Temperature PV*)
a7_dataLink[15].sValue:=INT_TO_STRING(ARiStnManualUSBtmAsv[7]);(*U/Sonic Bottom A Power SV*)
a7_dataLink[16].sValue:=INT_TO_STRING(ARiStnUSBtmAPv[7]);(*U/Sonic Bottom A Power PV*)
a7_dataLink[17].sValue:='N/A';(*U/Sonic Bottom A Frequency SV*)
a7_dataLink[18].sValue:=INT_TO_STRING(DSWeberEnclosure[1].DSWeberGenerator[7].IN_iFreqSetPoint);(*U/Sonic Bottom A Frequency PV*)
a7_dataLink[19].sValue:=INT_TO_STRING(ARiStnManualUSBtmBsv[7]);(*U/Sonic Bottom B Power SV*)
a7_dataLink[20].sValue:=INT_TO_STRING(ARiStnUSBtmBPv[7]);(*U/Sonic Bottom B Power PV*)
a7_dataLink[21].sValue:='N/A';(*U/Sonic Bottom B Frequency SV*)
a7_dataLink[22].sValue:='N/A';(*U/Sonic Bottom B Frequency PV*)
a7_dataLink[23].sValue:='N/A';(*U/Sonic Side A Power SV*)
a7_dataLink[24].sValue:='N/A';(*U/Sonic Side A Power PV*)
a7_dataLink[25].sValue:='N/A';(*U/Sonic Side A Frequency SV*)
a7_dataLink[26].sValue:='N/A';(*U/Sonic Side A Frequency PV*)
a7_dataLink[27].sValue:='N/A';(*U/Sonic Side B Power SV*)
a7_dataLink[28].sValue:='N/A';(*U/Sonic Side B Power PV*)
a7_dataLink[29].sValue:='N/A';(*U/Sonic Side B Frequency SV*)
a7_dataLink[30].sValue:='N/A';(*U/Sonic Side B Frequency PV*)
a7_dataLink[31].sValue:='N/A';(*Vacuum SV*)
a7_dataLink[32].sValue:='N/A';(*Vacuum PV*)
a7_dataLink[33].sValue:='N/A';(*Conductivity SV*)
a7_dataLink[34].sValue:=REAL_TO_STRING(ARrStnConductivityPV[7]);(*Conductivity PV*)
a7_dataLink[35].sValue:='N/A';(*Pump Flow SV*)
a7_dataLink[36].sValue:=REAL_TO_STRING(ARrStnFilterPressurePV[7]);(*Pump Flow PV*)
a7_dataLink[37].sValue:='N/A';(*Resistivity SV*)
a7_dataLink[38].sValue:='N/A';(*Resistivity PV*)
a7_dataLink[39].sValue:='N/A';(*PH SV*)
a7_dataLink[40].sValue:='N/A'; (*PH PV*)
a7_dataLink[41].sValue:='N/A';(*Quality*)
a7_dataLink[42].sValue:=DSStnBasketInfo[7].sProductQuality;(*Quality*)
a7_dataLink[43].sValue:=INT_TO_STRING(ARDsStnSeqProcessCtrl[7].Out_iCurrentProcessTime);(*Actual Time*)
a7_dataLink[44].sValue:='N/A';(*Actual Time*)

(************************************************************************************************************************)

a8_dataLink[1].sName4:='';
a8_dataLink[2].sName4:='Operator';
a8_dataLink[3].sName4:='LD ID';
a8_dataLink[4].sName4:='ULD ID';
a8_dataLink[5].sName4:='Pro Recipe No';
a8_dataLink[6].sName4:='Pro Recipe Dscrp';
a8_dataLink[7].sName4:='LD No';


a8_dataLink[1].sName3:='';
a8_dataLink[2].sName3:=sUserName;
a8_dataLink[3].sName3:='1';
a8_dataLink[4].sName3:='1';
a8_dataLink[5].sName3:=INT_TO_STRING(DSStnBasketInfo[8].iProductRecipeNo);
a8_dataLink[6].sName3:=DSStnBasketInfo[8].sProgramDescription;
a8_dataLink[7].sName3:=INT_TO_STRING(iProgBatchTotal);


a8_dataLink[1].sName2:='';
a8_dataLink[2].sName2:='N/A';
a8_dataLink[3].sName2:='N/A';
a8_dataLink[4].sName2:='N/A';
a8_dataLink[5].sName2:='N/A';
a8_dataLink[6].sName2:='N/A';
a8_dataLink[7].sName2:='N/A';
a8_dataLink[8].sName2:='Sec';
a8_dataLink[9].sName2:='Sec';
a8_dataLink[10].sName2:='Sec';
a8_dataLink[11].sName2:='Sec';
a8_dataLink[12].sName2:='Sec';
a8_dataLink[13].sName2:='Sec';
a8_dataLink[14].sName2:='DegC';
a8_dataLink[15].sName2:='DegC';
a8_dataLink[16].sName2:='%';
a8_dataLink[17].sName2:='%';
a8_dataLink[18].sName2:='Hz';
a8_dataLink[19].sName2:='Hz';
a8_dataLink[20].sName2:='%';
a8_dataLink[21].sName2:='%';
a8_dataLink[22].sName2:='Hz';
a8_dataLink[23].sName2:='Hz';
a8_dataLink[24].sName2:='%';
a8_dataLink[25].sName2:='%';
a8_dataLink[26].sName2:='Hz';
a8_dataLink[27].sName2:='Hz';
a8_dataLink[28].sName2:='%';
a8_dataLink[29].sName2:='%';
a8_dataLink[30].sName2:='Hz';
a8_dataLink[31].sName2:='Hz';
a8_dataLink[32].sName2:='Kpa';
a8_dataLink[33].sName2:='Kpa';
a8_dataLink[34].sName2:='uS';
a8_dataLink[35].sName2:='uS';
a8_dataLink[36].sName2:='LPM';
a8_dataLink[37].sName2:='LPM';
a8_dataLink[38].sName2:='OHM';
a8_dataLink[39].sName2:='OHM';
a8_dataLink[40].sName2:='PH';
a8_dataLink[41].sName2:='PH';
a8_dataLink[42].sName2:='N/A';
a8_dataLink[43].sName2:='N/A';
a8_dataLink[44].sName2:='Sec';
a8_dataLink[45].sName2:='Sec';



a8_dataLink[1].sName:='Station';
a8_dataLink[2].sName:='Station';
a8_dataLink[3].sName:='Sequences Recipe';
a8_dataLink[4].sName:='Sequences Recipe';
a8_dataLink[5].sName:='Sub Recipe';
a8_dataLink[6].sName:='Sub Recipe';
a8_dataLink[7].sName:='Minimum Time';
a8_dataLink[8].sName:='Minimum Time';
a8_dataLink[9].sName:='Maximum Time';
a8_dataLink[10].sName:='Maximum Time';
a8_dataLink[11].sName:='Effective Time';
a8_dataLink[12].sName:='Effective Time';
a8_dataLink[13].sName:='Temperature';
a8_dataLink[14].sName:='Temperature';
a8_dataLink[15].sName:='U/Sonic Bottom A Power';
a8_dataLink[16].sName:='U/Sonic Bottom A Power';
a8_dataLink[17].sName:='U/Sonic Bottom A Frequency';
a8_dataLink[18].sName:='U/Sonic Bottom A Frequency';
a8_dataLink[19].sName:='U/Sonic Bottom B Power';
a8_dataLink[20].sName:='U/Sonic Bottom B Power';
a8_dataLink[21].sName:='U/Sonic Bottom B Frequency';
a8_dataLink[22].sName:='U/Sonic Bottom B Frequency';
a8_dataLink[23].sName:='U/Sonic Side A Power SV';
a8_dataLink[24].sName:='U/Sonic Side A Power PV';
a8_dataLink[25].sName:='U/Sonic Side A Frequency';
a8_dataLink[26].sName:='U/Sonic Side A Frequency';
a8_dataLink[27].sName:='U/Sonic Side B Power';
a8_dataLink[28].sName:='U/Sonic Side B Power';
a8_dataLink[29].sName:='U/Sonic Side B Frequency';
a8_dataLink[30].sName:='U/Sonic Side B Frequency';
a8_dataLink[31].sName:='Vacuum SV';
a8_dataLink[32].sName:='Vacuum PV';
a8_dataLink[33].sName:='Conductivity';
a8_dataLink[34].sName:='Conductivity';
a8_dataLink[35].sName:='Pump Flow';
a8_dataLink[36].sName:='Pump Flow';
a8_dataLink[37].sName:='Resistivity';
a8_dataLink[38].sName:='Resistivity';
a8_dataLink[39].sName:='PH PV';
a8_dataLink[40].sName:='PH PV';
a8_dataLink[41].sName:='Quality';
a8_dataLink[42].sName:='Quality';
a8_dataLink[43].sName:='Actual Time';
a8_dataLink[44].sName:='Actual Time';


a8_dataLink[1].sValue:='N/A';(*Station*)
a8_dataLink[2].sValue:='8-Rinsing DI Water';(*Station*)
a8_dataLink[3].sValue:='N/A';(*Sequences Recipe*)
a8_dataLink[4].sValue:=DSHmiStationDisplayInfo[8].sStationSequenceRecipeDescription;(*Sequences Recipe*)
a8_dataLink[5].sValue:='N/A';(*Sub Recipe*)
a8_dataLink[6].sValue:=DSHmiStationDisplayInfo[8].sStationSubDescription;(*Sub Recipe*)
a8_dataLink[7].sValue:=INT_TO_STRING(ARDsStnMinMaxEffTimeDisplay[8].iMinTime);(*Minimum Time*)
a8_dataLink[8].sValue:='N/A';(*Minimum Time*)
a8_dataLink[9].sValue:=INT_TO_STRING(ARDsStnMinMaxEffTimeDisplay[8].iMaxTime);(*Maximum Time*)
a8_dataLink[10].sValue:='N/A';(*Maximum Time*)
a8_dataLink[11].sValue:=INT_TO_STRING(ARDsStnMinMaxEffTimeDisplay[8].iEffTime);(*Effective Time*)
a8_dataLink[12].sValue:='N/A';(*Effective Time*)
a8_dataLink[13].sValue:=REAL_TO_STRING(ARrStnTempSV[8]);(*Temperature SV*)
a8_dataLink[14].sValue:=REAL_TO_STRING(ARrStnTempPV[8]);(*Temperature PV*)
a8_dataLink[15].sValue:=INT_TO_STRING(ARiStnManualUSBtmAsv[8]);(*U/Sonic Bottom A Power SV*)
a8_dataLink[16].sValue:=INT_TO_STRING(ARiStnUSBtmAPv[8]);(*U/Sonic Bottom A Power PV*)
a8_dataLink[17].sValue:='N/A';(*U/Sonic Bottom A Frequency SV*)
a8_dataLink[18].sValue:='N/A';(*U/Sonic Bottom A Frequency PV*)
a8_dataLink[19].sValue:=INT_TO_STRING(ARiStnManualUSBtmBsv[8]);(*U/Sonic Bottom B Power SV*)
a8_dataLink[20].sValue:=INT_TO_STRING(ARiStnUSBtmBPv[8]);(*U/Sonic Bottom B Power PV*)
a8_dataLink[21].sValue:='N/A';(*U/Sonic Bottom B Frequency SV*)
a8_dataLink[22].sValue:='N/A';(*U/Sonic Bottom B Frequency PV*)
a8_dataLink[23].sValue:='N/A';(*U/Sonic Side A Power SV*)
a8_dataLink[24].sValue:='N/A';(*U/Sonic Side A Power PV*)
a8_dataLink[25].sValue:='N/A';(*U/Sonic Side A Frequency SV*)
a8_dataLink[26].sValue:='N/A';(*U/Sonic Side A Frequency PV*)
a8_dataLink[27].sValue:='N/A';(*U/Sonic Side B Power SV*)
a8_dataLink[28].sValue:='N/A';(*U/Sonic Side B Power PV*)
a8_dataLink[29].sValue:='N/A';(*U/Sonic Side B Frequency SV*)
a8_dataLink[30].sValue:='N/A';(*U/Sonic Side B Frequency PV*)
a8_dataLink[31].sValue:='N/A';(*Vacuum SV*)
a8_dataLink[32].sValue:='N/A';(*Vacuum PV*)
a8_dataLink[33].sValue:='N/A';(*Conductivity SV*)
a8_dataLink[34].sValue:=REAL_TO_STRING(ARrStnConductivityPV[8]);(*Conductivity PV*)
a8_dataLink[35].sValue:='N/A';(*Pump Flow SV*)
a8_dataLink[36].sValue:=REAL_TO_STRING(ARrStnFilterPressurePV[8]);(*Pump Flow PV*)
a8_dataLink[37].sValue:='N/A';(*Resistivity SV*)
a8_dataLink[38].sValue:='N/A';(*Resistivity PV*)
a8_dataLink[39].sValue:='N/A';(*PH SV*)
a8_dataLink[40].sValue:='N/A'; (*PH PV*)
a8_dataLink[41].sValue:='N/A';(*Quality*)
a8_dataLink[42].sValue:=DSStnBasketInfo[8].sProductQuality;(*Quality*)
a8_dataLink[43].sValue:=INT_TO_STRING(ARDsStnSeqProcessCtrl[8].Out_iCurrentProcessTime);(*Actual Time*)
a8_dataLink[44].sValue:='N/A';(*Actual Time*)


(************************************************************************************************************************)
a9_dataLink[1].sName4:='';
a9_dataLink[2].sName4:='Operator';
a9_dataLink[3].sName4:='LD ID';
a9_dataLink[4].sName4:='ULD ID';
a9_dataLink[5].sName4:='Pro Recipe No';
a9_dataLink[6].sName4:='Pro Recipe Dscrp';
a9_dataLink[7].sName4:='LD No';


a9_dataLink[1].sName3:='';
a9_dataLink[2].sName3:=sUserName;
a9_dataLink[3].sName3:='1';
a9_dataLink[4].sName3:='1';
a9_dataLink[5].sName3:=INT_TO_STRING(DSStnBasketInfo[9].iProductRecipeNo);
a9_dataLink[6].sName3:=DSStnBasketInfo[9].sProgramDescription;
a9_dataLink[7].sName3:=INT_TO_STRING(iProgBatchTotal);

a9_dataLink[1].sName2:='';
a9_dataLink[2].sName2:='N/A';
a9_dataLink[3].sName2:='N/A';
a9_dataLink[4].sName2:='N/A';
a9_dataLink[5].sName2:='N/A';
a9_dataLink[6].sName2:='N/A';
a9_dataLink[7].sName2:='N/A';
a9_dataLink[8].sName2:='Sec';
a9_dataLink[9].sName2:='Sec';
a9_dataLink[10].sName2:='Sec';
a9_dataLink[11].sName2:='Sec';
a9_dataLink[12].sName2:='Sec';
a9_dataLink[13].sName2:='Sec';
a9_dataLink[14].sName2:='DegC';
a9_dataLink[15].sName2:='DegC';
a9_dataLink[16].sName2:='%';
a9_dataLink[17].sName2:='%';
a9_dataLink[18].sName2:='Hz';
a9_dataLink[19].sName2:='Hz';
a9_dataLink[20].sName2:='%';
a9_dataLink[21].sName2:='%';
a9_dataLink[22].sName2:='Hz';
a9_dataLink[23].sName2:='Hz';
a9_dataLink[24].sName2:='%';
a9_dataLink[25].sName2:='%';
a9_dataLink[26].sName2:='Hz';
a9_dataLink[27].sName2:='Hz';
a9_dataLink[28].sName2:='%';
a9_dataLink[29].sName2:='%';
a9_dataLink[30].sName2:='Hz';
a9_dataLink[31].sName2:='Hz';
a9_dataLink[32].sName2:='Kpa';
a9_dataLink[33].sName2:='Kpa';
a9_dataLink[34].sName2:='uS';
a9_dataLink[35].sName2:='uS';
a9_dataLink[36].sName2:='LPM';
a9_dataLink[37].sName2:='LPM';
a9_dataLink[38].sName2:='OHM';
a9_dataLink[39].sName2:='OHM';
a9_dataLink[40].sName2:='PH';
a9_dataLink[41].sName2:='PH';
a9_dataLink[42].sName2:='N/A';
a9_dataLink[43].sName2:='N/A';
a9_dataLink[44].sName2:='Sec';
a9_dataLink[45].sName2:='Sec';

a9_dataLink[1].sName:='Station';
a9_dataLink[2].sName:='Station';
a9_dataLink[3].sName:='Sequences Recipe';
a9_dataLink[4].sName:='Sequences Recipe';
a9_dataLink[5].sName:='Sub Recipe';
a9_dataLink[6].sName:='Sub Recipe';
a9_dataLink[7].sName:='Minimum Time';
a9_dataLink[8].sName:='Minimum Time';
a9_dataLink[9].sName:='Maximum Time';
a9_dataLink[10].sName:='Maximum Time';
a9_dataLink[11].sName:='Effective Time';
a9_dataLink[12].sName:='Effective Time';
a9_dataLink[13].sName:='Temperature';
a9_dataLink[14].sName:='Temperature';
a9_dataLink[15].sName:='U/Sonic Bottom A Power';
a9_dataLink[16].sName:='U/Sonic Bottom A Power';
a9_dataLink[17].sName:='U/Sonic Bottom A Frequency';
a9_dataLink[18].sName:='U/Sonic Bottom A Frequency';
a9_dataLink[19].sName:='U/Sonic Bottom B Power';
a9_dataLink[20].sName:='U/Sonic Bottom B Power';
a9_dataLink[21].sName:='U/Sonic Bottom B Frequency';
a9_dataLink[22].sName:='U/Sonic Bottom B Frequency';
a9_dataLink[23].sName:='U/Sonic Side A Power SV';
a9_dataLink[24].sName:='U/Sonic Side A Power PV';
a9_dataLink[25].sName:='U/Sonic Side A Frequency';
a9_dataLink[26].sName:='U/Sonic Side A Frequency';
a9_dataLink[27].sName:='U/Sonic Side B Power';
a9_dataLink[28].sName:='U/Sonic Side B Power';
a9_dataLink[29].sName:='U/Sonic Side B Frequency';
a9_dataLink[30].sName:='U/Sonic Side B Frequency';
a9_dataLink[31].sName:='Vacuum SV';
a9_dataLink[32].sName:='Vacuum PV';
a9_dataLink[33].sName:='Conductivity';
a9_dataLink[34].sName:='Conductivity';
a9_dataLink[35].sName:='Pump Flow';
a9_dataLink[36].sName:='Pump Flow';
a9_dataLink[37].sName:='Resistivity';
a9_dataLink[38].sName:='Resistivity';
a9_dataLink[39].sName:='PH PV';
a9_dataLink[40].sName:='PH PV';
a9_dataLink[41].sName:='Quality';
a9_dataLink[42].sName:='Quality';
a9_dataLink[43].sName:='Actual Time';
a9_dataLink[44].sName:='Actual Time';

a9_dataLink[1].sValue:='N/A';(*Station*)
a9_dataLink[2].sValue:='9-Hot Air Drying';(*Station*)
a9_dataLink[3].sValue:='N/A';(*Sequences Recipe*)
a9_dataLink[4].sValue:=DSHmiStationDisplayInfo[9].sStationSequenceRecipeDescription;(*Sequences Recipe*)
a9_dataLink[5].sValue:='N/A';(*Sub Recipe*)
a9_dataLink[6].sValue:=DSHmiStationDisplayInfo[9].sStationSubDescription;(*Sub Recipe*)
a9_dataLink[7].sValue:=INT_TO_STRING(ARDsStnMinMaxEffTimeDisplay[9].iMinTime);(*Minimum Time*)
a9_dataLink[8].sValue:='N/A';(*Minimum Time*)
a9_dataLink[9].sValue:=INT_TO_STRING(ARDsStnMinMaxEffTimeDisplay[9].iMaxTime);(*Maximum Time*)
a9_dataLink[10].sValue:='N/A';(*Maximum Time*)
a9_dataLink[11].sValue:=INT_TO_STRING(ARDsStnMinMaxEffTimeDisplay[9].iEffTime);(*Effective Time*)
a9_dataLink[12].sValue:='N/A';(*Effective Time*)
a9_dataLink[13].sValue:=REAL_TO_STRING(ARrStnTempSV[9]);(*Temperature SV*)
a9_dataLink[14].sValue:=REAL_TO_STRING(ARrStnTempPV[9]);(*Temperature PV*)
a9_dataLink[15].sValue:=INT_TO_STRING(ARiStnManualUSBtmAsv[9]);(*U/Sonic Bottom A Power SV*)
a9_dataLink[16].sValue:=INT_TO_STRING(ARiStnUSBtmAPv[9]);(*U/Sonic Bottom A Power PV*)
a9_dataLink[17].sValue:='N/A';(*U/Sonic Bottom A Frequency SV*)
a9_dataLink[18].sValue:='N/A';(*U/Sonic Bottom A Frequency PV*)
a9_dataLink[19].sValue:=INT_TO_STRING(ARiStnManualUSBtmBsv[9]);(*U/Sonic Bottom B Power SV*)
a9_dataLink[20].sValue:=INT_TO_STRING(ARiStnUSBtmBPv[9]);(*U/Sonic Bottom B Power PV*)
a9_dataLink[21].sValue:='N/A';(*U/Sonic Bottom B Frequency SV*)
a9_dataLink[22].sValue:='N/A';(*U/Sonic Bottom B Frequency PV*)
a9_dataLink[23].sValue:='N/A';(*U/Sonic Side A Power SV*)
a9_dataLink[24].sValue:='N/A';(*U/Sonic Side A Power PV*)
a9_dataLink[25].sValue:='N/A';(*U/Sonic Side A Frequency SV*)
a9_dataLink[26].sValue:='N/A';(*U/Sonic Side A Frequency PV*)
a9_dataLink[27].sValue:='N/A';(*U/Sonic Side B Power SV*)
a9_dataLink[28].sValue:='N/A';(*U/Sonic Side B Power PV*)
a9_dataLink[29].sValue:='N/A';(*U/Sonic Side B Frequency SV*)
a9_dataLink[30].sValue:='N/A';(*U/Sonic Side B Frequency PV*)
a9_dataLink[31].sValue:='N/A';(*Vacuum SV*)
a9_dataLink[32].sValue:='N/A';(*Vacuum PV*)
a9_dataLink[33].sValue:='N/A';(*Conductivity SV*)
a9_dataLink[34].sValue:=REAL_TO_STRING(ARrStnConductivityPV[9]);(*Conductivity PV*)
a9_dataLink[35].sValue:='N/A';(*Pump Flow SV*)
a9_dataLink[36].sValue:=REAL_TO_STRING(ARrStnFilterPressurePV[9]);(*Pump Flow PV*)
a9_dataLink[37].sValue:='N/A';(*Resistivity SV*)
a9_dataLink[38].sValue:='N/A';(*Resistivity PV*)
a9_dataLink[39].sValue:='N/A';(*PH SV*)
a9_dataLink[40].sValue:='N/A'; (*PH PV*)
a9_dataLink[41].sValue:='N/A';(*Quality*)
a9_dataLink[42].sValue:=DSStnBasketInfo[9].sProductQuality;(*Quality*)
a9_dataLink[43].sValue:=INT_TO_STRING(ARDsStnSeqProcessCtrl[9].Out_iCurrentProcessTime);(*Actual Time*)
a9_dataLink[44].sValue:='N/A';(*Actual Time*)

(************************************************************************************************************************)
a10_dataLink[1].sName4:='';
a10_dataLink[2].sName4:='Operator';
a10_dataLink[3].sName4:='LD ID';
a10_dataLink[4].sName4:='ULD ID';
a10_dataLink[5].sName4:='Pro Recipe No';
a10_dataLink[6].sName4:='Pro Recipe Dscrp';
a10_dataLink[7].sName4:='LD No';


a10_dataLink[1].sName3:='';
a10_dataLink[2].sName3:=sUserName;
a10_dataLink[3].sName3:='1';
a10_dataLink[4].sName3:='1';
a10_dataLink[5].sName3:=INT_TO_STRING(DSStnBasketInfo[10].iProductRecipeNo);
a10_dataLink[6].sName3:=DSStnBasketInfo[10].sProgramDescription;
a10_dataLink[7].sName3:=INT_TO_STRING(iProgBatchTotal);

a10_dataLink[1].sName2:='';
a10_dataLink[2].sName2:='N/A';
a10_dataLink[3].sName2:='N/A';
a10_dataLink[4].sName2:='N/A';
a10_dataLink[5].sName2:='N/A';
a10_dataLink[6].sName2:='N/A';
a10_dataLink[7].sName2:='N/A';
a10_dataLink[8].sName2:='Sec';
a10_dataLink[9].sName2:='Sec';
a10_dataLink[10].sName2:='Sec';
a10_dataLink[11].sName2:='Sec';
a10_dataLink[12].sName2:='Sec';
a10_dataLink[13].sName2:='Sec';
a10_dataLink[14].sName2:='DegC';
a10_dataLink[15].sName2:='DegC';
a10_dataLink[16].sName2:='%';
a10_dataLink[17].sName2:='%';
a10_dataLink[18].sName2:='Hz';
a10_dataLink[19].sName2:='Hz';
a10_dataLink[20].sName2:='%';
a10_dataLink[21].sName2:='%';
a10_dataLink[22].sName2:='Hz';
a10_dataLink[23].sName2:='Hz';
a10_dataLink[24].sName2:='%';
a10_dataLink[25].sName2:='%';
a10_dataLink[26].sName2:='Hz';
a10_dataLink[27].sName2:='Hz';
a10_dataLink[28].sName2:='%';
a10_dataLink[29].sName2:='%';
a10_dataLink[30].sName2:='Hz';
a10_dataLink[31].sName2:='Hz';
a10_dataLink[32].sName2:='Kpa';
a10_dataLink[33].sName2:='Kpa';
a10_dataLink[34].sName2:='uS';
a10_dataLink[35].sName2:='uS';
a10_dataLink[36].sName2:='LPM';
a10_dataLink[37].sName2:='LPM';
a10_dataLink[38].sName2:='OHM';
a10_dataLink[39].sName2:='OHM';
a10_dataLink[40].sName2:='PH';
a10_dataLink[41].sName2:='PH';
a10_dataLink[42].sName2:='N/A';
a10_dataLink[43].sName2:='N/A';
a10_dataLink[44].sName2:='Sec';
a10_dataLink[45].sName2:='Sec';

